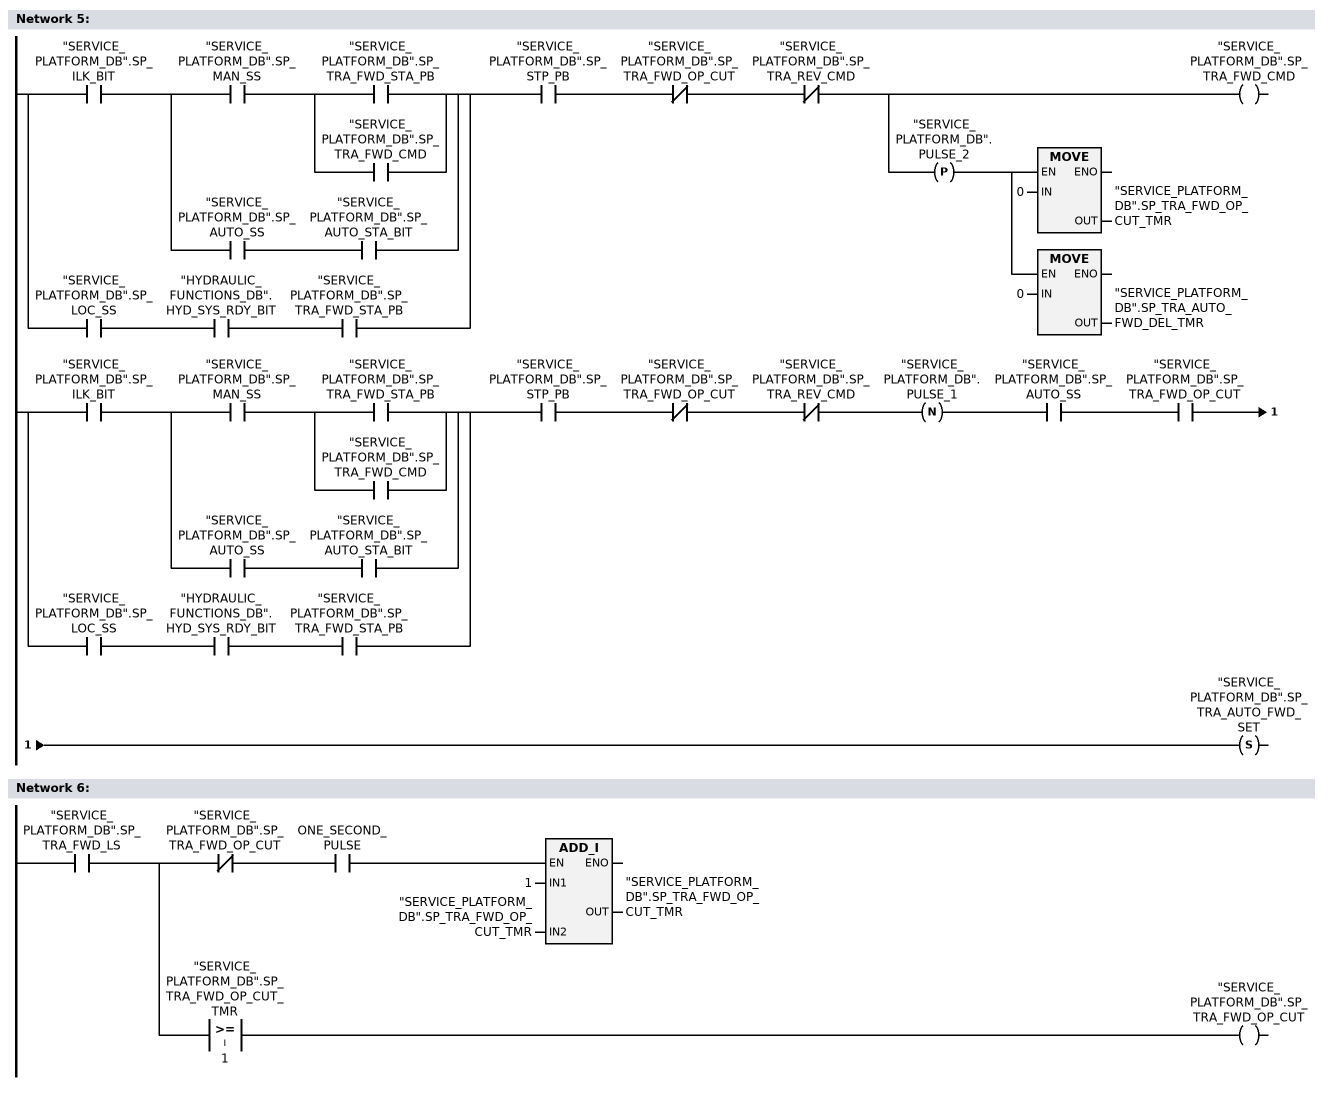
NETWORK
TITLE =
      A(;
      A     "SERVICE_PLATFORM_DB".SP_ILK_BIT;
      A(;
      A     "SERVICE_PLATFORM_DB".SP_MAN_SS;
      A(;
      O     "SERVICE_PLATFORM_DB".SP_TRA_FWD_STA_PB;
      O     "SERVICE_PLATFORM_DB".SP_TRA_FWD_CMD;
      );
      O;
      A     "SERVICE_PLATFORM_DB".SP_AUTO_SS;
      A     "SERVICE_PLATFORM_DB".SP_AUTO_STA_BIT;
      );
      O;
      A     "SERVICE_PLATFORM_DB".SP_LOC_SS;
      A     "HYDRAULIC_FUNCTIONS_DB".HYD_SYS_RDY_BIT;
      A     "SERVICE_PLATFORM_DB".SP_TRA_FWD_STA_PB;
      );
      A     "SERVICE_PLATFORM_DB".SP_STP_PB;
      AN    "SERVICE_PLATFORM_DB".SP_TRA_FWD_OP_CUT;
      AN    "SERVICE_PLATFORM_DB".SP_TRA_REV_CMD;
      =     L 0.0;
      A     L 0.0;
      BLD   102;
      =     "SERVICE_PLATFORM_DB".SP_TRA_FWD_CMD;
      A(;
      A     L 0.0;
      FN    "SERVICE_PLATFORM_DB".PULSE_1;
      );
      A     "SERVICE_PLATFORM_DB".SP_AUTO_SS;
      A     "SERVICE_PLATFORM_DB".SP_TRA_FWD_OP_CUT;
      S     "SERVICE_PLATFORM_DB".SP_TRA_AUTO_FWD_SET;
      A     L 0.0;
      FP    "SERVICE_PLATFORM_DB".PULSE_2;
      =     L 0.1;
      A     L 0.1;
      JNB   M001;
      L     0;
      T     "SERVICE_PLATFORM_DB".SP_TRA_FWD_OP_CUT_TMR;
M001: NOP   0;
      A     L 0.1;
      JNB   M002;
      L     0;
      T     "SERVICE_PLATFORM_DB".SP_TRA_AUTO_FWD_DEL_TMR;
M002: NOP   0;
NETWORK
TITLE =
      A     "SERVICE_PLATFORM_DB".SP_TRA_FWD_LS;
      =     L 0.0;
      A     L 0.0;
      AN    "SERVICE_PLATFORM_DB".SP_TRA_FWD_OP_CUT;
      A     "ONE_SECOND_PULSE";
      JNB   M003;
      L     1;
      L     "SERVICE_PLATFORM_DB".SP_TRA_FWD_OP_CUT_TMR;
      +I;
      T     "SERVICE_PLATFORM_DB".SP_TRA_FWD_OP_CUT_TMR;
M003: NOP   0;
      A     L 0.0;
      A(;
      L     "SERVICE_PLATFORM_DB".SP_TRA_FWD_OP_CUT_TMR;
      L     1;
      >=I;
      );
      =     "SERVICE_PLATFORM_DB".SP_TRA_FWD_OP_CUT;
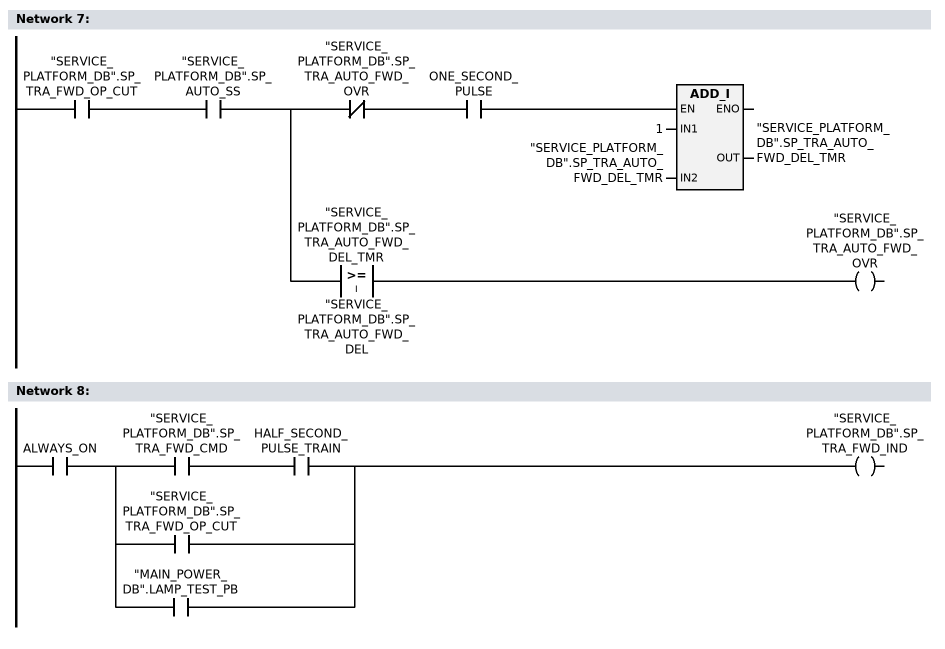
NETWORK
TITLE =
      A     "SERVICE_PLATFORM_DB".SP_TRA_FWD_OP_CUT;
      A     "SERVICE_PLATFORM_DB".SP_AUTO_SS;
      =     L 0.0;
      A     L 0.0;
      AN    "SERVICE_PLATFORM_DB".SP_TRA_AUTO_FWD_OVR;
      A     "ONE_SECOND_PULSE";
      JNB   M004;
      L     1;
      L     "SERVICE_PLATFORM_DB".SP_TRA_AUTO_FWD_DEL_TMR;
      +I;
      T     "SERVICE_PLATFORM_DB".SP_TRA_AUTO_FWD_DEL_TMR;
M004: NOP   0;
      A     L 0.0;
      A(;
      L     "SERVICE_PLATFORM_DB".SP_TRA_AUTO_FWD_DEL_TMR;
      L     "SERVICE_PLATFORM_DB".SP_TRA_AUTO_FWD_DEL;
      >=I;
      );
      =     "SERVICE_PLATFORM_DB".SP_TRA_AUTO_FWD_OVR;
NETWORK
TITLE =
      A     "ALWAYS_ON";
      A(;
      A     "SERVICE_PLATFORM_DB".SP_TRA_FWD_CMD;
      A     "HALF_SECOND_PULSE_TRAIN";
      O     "SERVICE_PLATFORM_DB".SP_TRA_FWD_OP_CUT;
      O     "MAIN_POWER_DB".LAMP_TEST_PB;
      );
      =     "SERVICE_PLATFORM_DB".SP_TRA_FWD_IND;
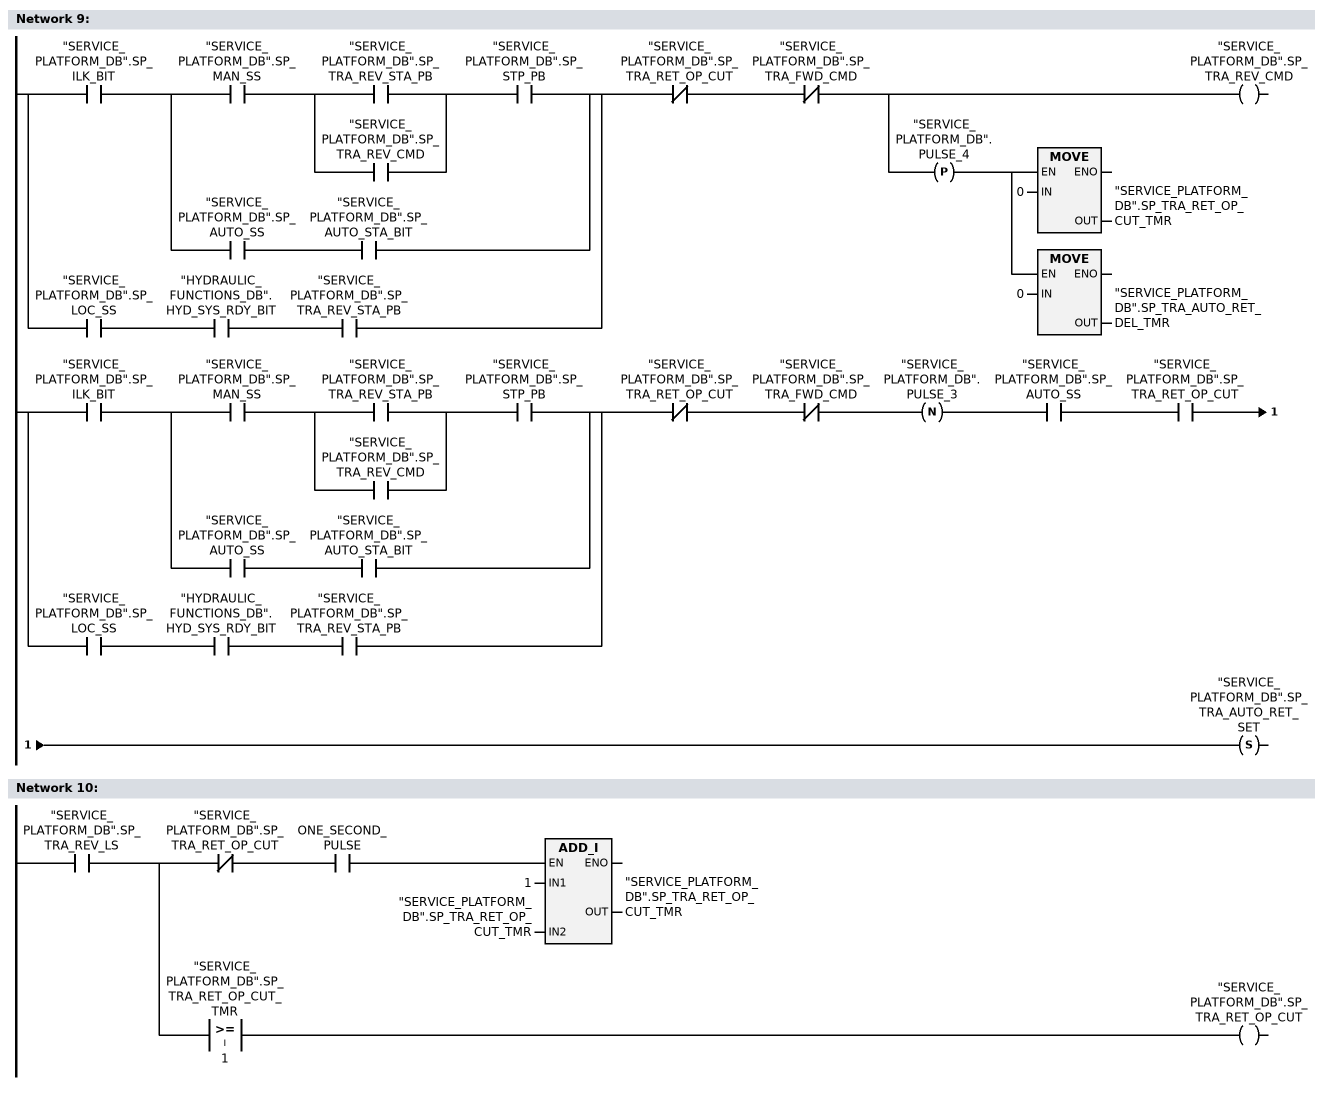
NETWORK
TITLE =
      A(;
      A     "SERVICE_PLATFORM_DB".SP_ILK_BIT;
      A(;
      A     "SERVICE_PLATFORM_DB".SP_MAN_SS;
      A(;
      O     "SERVICE_PLATFORM_DB".SP_TRA_REV_STA_PB;
      O     "SERVICE_PLATFORM_DB".SP_TRA_REV_CMD;
      );
      A     "SERVICE_PLATFORM_DB".SP_STP_PB;
      O;
      A     "SERVICE_PLATFORM_DB".SP_AUTO_SS;
      A     "SERVICE_PLATFORM_DB".SP_AUTO_STA_BIT;
      );
      O;
      A     "SERVICE_PLATFORM_DB".SP_LOC_SS;
      A     "HYDRAULIC_FUNCTIONS_DB".HYD_SYS_RDY_BIT;
      A     "SERVICE_PLATFORM_DB".SP_TRA_REV_STA_PB;
      );
      AN    "SERVICE_PLATFORM_DB".SP_TRA_RET_OP_CUT;
      AN    "SERVICE_PLATFORM_DB".SP_TRA_FWD_CMD;
      =     L 0.0;
      A     L 0.0;
      BLD   102;
      =     "SERVICE_PLATFORM_DB".SP_TRA_REV_CMD;
      A(;
      A     L 0.0;
      FN    "SERVICE_PLATFORM_DB".PULSE_3;
      );
      A     "SERVICE_PLATFORM_DB".SP_AUTO_SS;
      A     "SERVICE_PLATFORM_DB".SP_TRA_RET_OP_CUT;
      S     "SERVICE_PLATFORM_DB".SP_TRA_AUTO_RET_SET;
      A     L 0.0;
      FP    "SERVICE_PLATFORM_DB".PULSE_4;
      =     L 0.1;
      A     L 0.1;
      JNB   M005;
      L     0;
      T     "SERVICE_PLATFORM_DB".SP_TRA_RET_OP_CUT_TMR;
M005: NOP   0;
      A     L 0.1;
      JNB   M006;
      L     0;
      T     "SERVICE_PLATFORM_DB".SP_TRA_AUTO_RET_DEL_TMR;
M006: NOP   0;
NETWORK
TITLE =
      A     "SERVICE_PLATFORM_DB".SP_TRA_REV_LS;
      =     L 0.0;
      A     L 0.0;
      AN    "SERVICE_PLATFORM_DB".SP_TRA_RET_OP_CUT;
      A     "ONE_SECOND_PULSE";
      JNB   M007;
      L     1;
      L     "SERVICE_PLATFORM_DB".SP_TRA_RET_OP_CUT_TMR;
      +I;
      T     "SERVICE_PLATFORM_DB".SP_TRA_RET_OP_CUT_TMR;
M007: NOP   0;
      A     L 0.0;
      A(;
      L     "SERVICE_PLATFORM_DB".SP_TRA_RET_OP_CUT_TMR;
      L     1;
      >=I;
      );
      =     "SERVICE_PLATFORM_DB".SP_TRA_RET_OP_CUT;
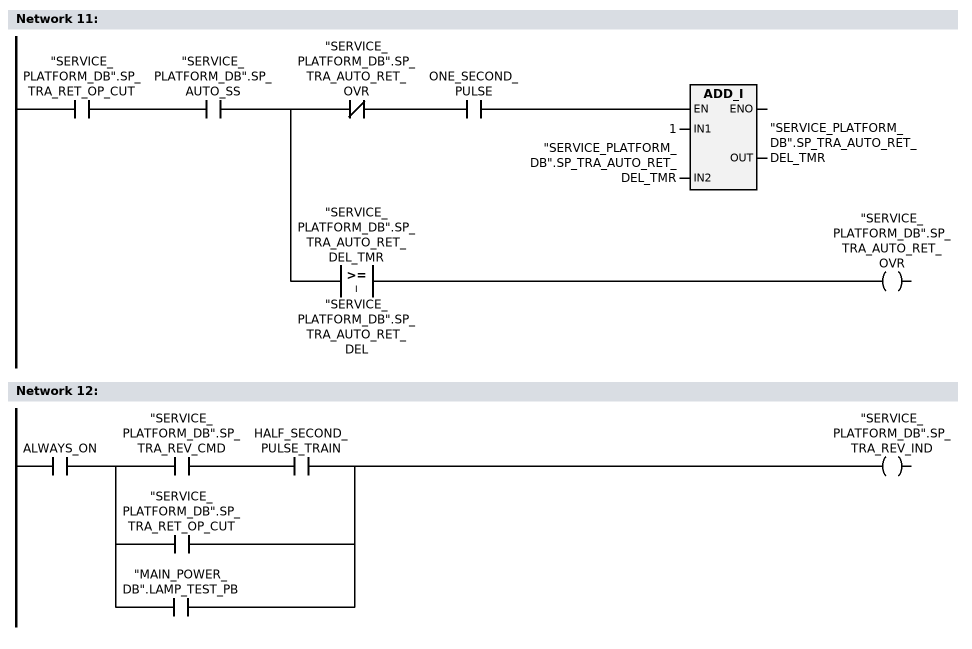
NETWORK
TITLE =
      A     "SERVICE_PLATFORM_DB".SP_TRA_RET_OP_CUT;
      A     "SERVICE_PLATFORM_DB".SP_AUTO_SS;
      =     L 0.0;
      A     L 0.0;
      AN    "SERVICE_PLATFORM_DB".SP_TRA_AUTO_RET_OVR;
      A     "ONE_SECOND_PULSE";
      JNB   M008;
      L     1;
      L     "SERVICE_PLATFORM_DB".SP_TRA_AUTO_RET_DEL_TMR;
      +I;
      T     "SERVICE_PLATFORM_DB".SP_TRA_AUTO_RET_DEL_TMR;
M008: NOP   0;
      A     L 0.0;
      A(;
      L     "SERVICE_PLATFORM_DB".SP_TRA_AUTO_RET_DEL_TMR;
      L     "SERVICE_PLATFORM_DB".SP_TRA_AUTO_RET_DEL;
      >=I;
      );
      =     "SERVICE_PLATFORM_DB".SP_TRA_AUTO_RET_OVR;
NETWORK
TITLE =
      A     "ALWAYS_ON";
      A(;
      A     "SERVICE_PLATFORM_DB".SP_TRA_REV_CMD;
      A     "HALF_SECOND_PULSE_TRAIN";
      O     "SERVICE_PLATFORM_DB".SP_TRA_RET_OP_CUT;
      O     "MAIN_POWER_DB".LAMP_TEST_PB;
      );
      =     "SERVICE_PLATFORM_DB".SP_TRA_REV_IND;
END_FUNCTION

FUNCTION "JAMB_CLEANER" : VOID	// FC 10
AUTHOR : Kamillas
VERSION : 0.1
BEGIN
// (block stored without names or comments; labels and parameter names are numbered)
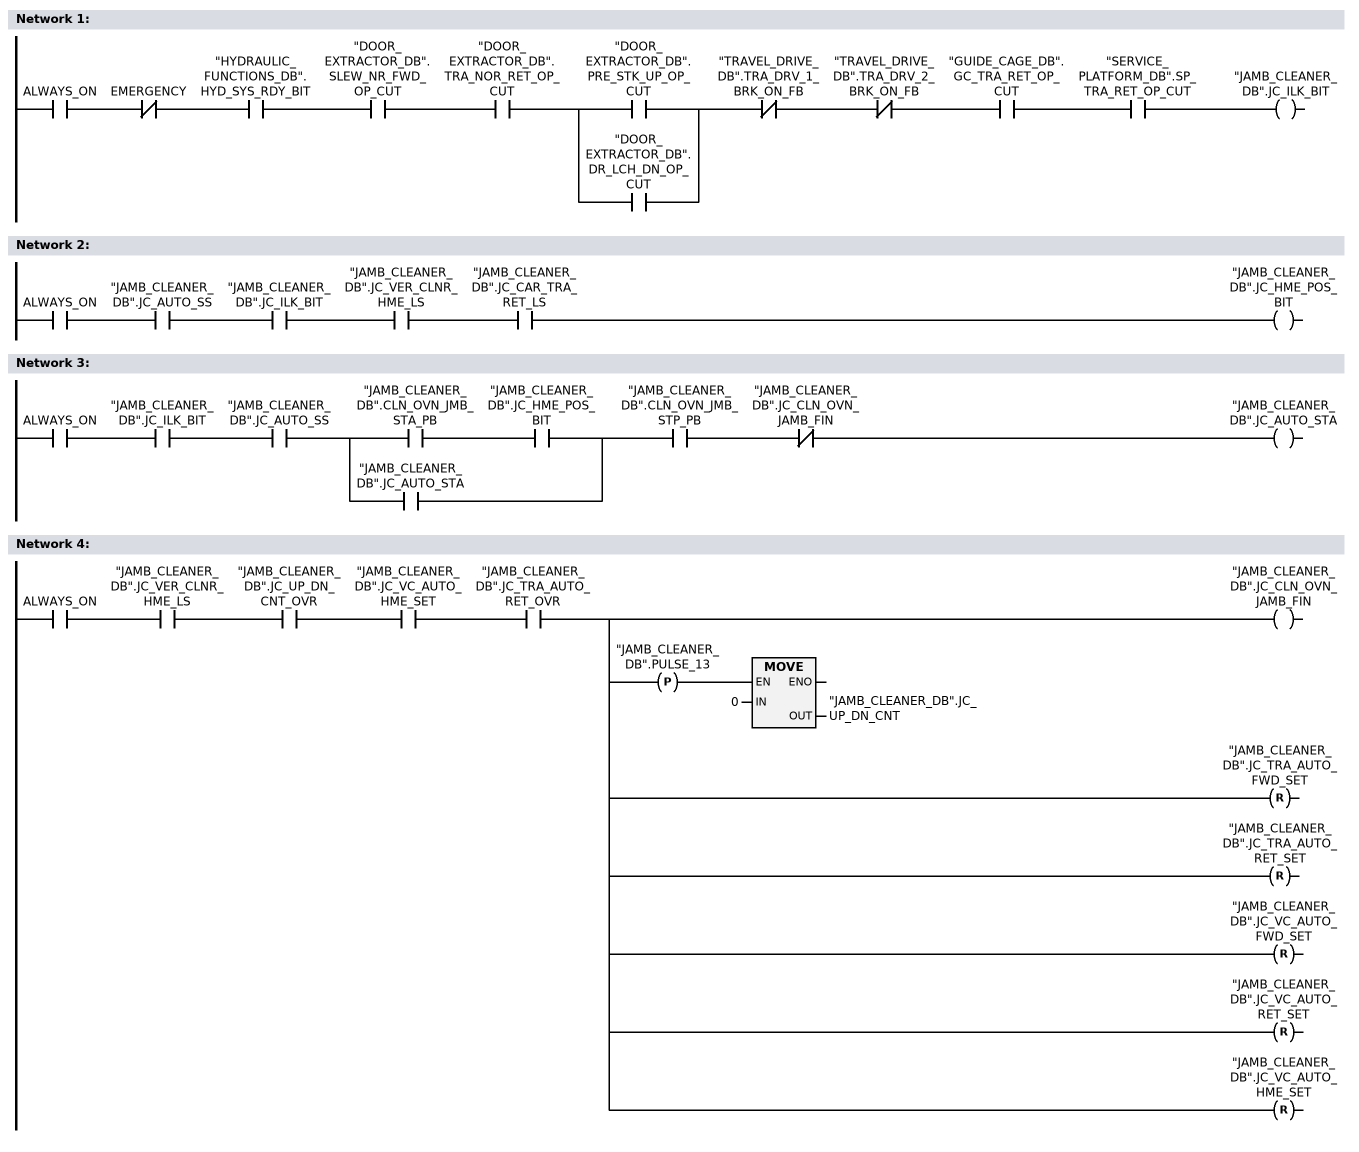
NETWORK
TITLE =
      A     "ALWAYS_ON";
      AN    "EMERGENCY";
      A     "HYDRAULIC_FUNCTIONS_DB".HYD_SYS_RDY_BIT;
      A     "DOOR_EXTRACTOR_DB".SLEW_NR_FWD_OP_CUT;
      A     "DOOR_EXTRACTOR_DB".TRA_NOR_RET_OP_CUT;
      A(;
      O     "DOOR_EXTRACTOR_DB".PRE_STK_UP_OP_CUT;
      O     "DOOR_EXTRACTOR_DB".DR_LCH_DN_OP_CUT;
      );
      AN    "TRAVEL_DRIVE_DB".TRA_DRV_1_BRK_ON_FB;
      AN    "TRAVEL_DRIVE_DB".TRA_DRV_2_BRK_ON_FB;
      A     "GUIDE_CAGE_DB".GC_TRA_RET_OP_CUT;
      A     "SERVICE_PLATFORM_DB".SP_TRA_RET_OP_CUT;
      =     "JAMB_CLEANER_DB".JC_ILK_BIT;
NETWORK
TITLE =
      A     "ALWAYS_ON";
      A     "JAMB_CLEANER_DB".JC_AUTO_SS;
      A     "JAMB_CLEANER_DB".JC_ILK_BIT;
      A     "JAMB_CLEANER_DB".JC_VER_CLNR_HME_LS;
      A     "JAMB_CLEANER_DB".JC_CAR_TRA_RET_LS;
      =     "JAMB_CLEANER_DB".JC_HME_POS_BIT;
NETWORK
TITLE =
      A     "ALWAYS_ON";
      A     "JAMB_CLEANER_DB".JC_ILK_BIT;
      A     "JAMB_CLEANER_DB".JC_AUTO_SS;
      A(;
      A     "JAMB_CLEANER_DB".CLN_OVN_JMB_STA_PB;
      A     "JAMB_CLEANER_DB".JC_HME_POS_BIT;
      O     "JAMB_CLEANER_DB".JC_AUTO_STA;
      );
      A     "JAMB_CLEANER_DB".CLN_OVN_JMB_STP_PB;
      AN    "JAMB_CLEANER_DB".JC_CLN_OVN_JAMB_FIN;
      =     "JAMB_CLEANER_DB".JC_AUTO_STA;
NETWORK
TITLE =
      A     "ALWAYS_ON";
      A     "JAMB_CLEANER_DB".JC_VER_CLNR_HME_LS;
      A     "JAMB_CLEANER_DB".JC_UP_DN_CNT_OVR;
      A     "JAMB_CLEANER_DB".JC_VC_AUTO_HME_SET;
      A     "JAMB_CLEANER_DB".JC_TRA_AUTO_RET_OVR;
      =     L 0.0;
      A     L 0.0;
      BLD   102;
      =     "JAMB_CLEANER_DB".JC_CLN_OVN_JAMB_FIN;
      A     L 0.0;
      FP    "JAMB_CLEANER_DB".PULSE_13;
      JNB   M001;
      L     0;
      T     "JAMB_CLEANER_DB".JC_UP_DN_CNT;
M001: NOP   0;
      A     L 0.0;
      BLD   102;
      R     "JAMB_CLEANER_DB".JC_TRA_AUTO_FWD_SET;
      A     L 0.0;
      BLD   102;
      R     "JAMB_CLEANER_DB".JC_TRA_AUTO_RET_SET;
      A     L 0.0;
      BLD   102;
      R     "JAMB_CLEANER_DB".JC_VC_AUTO_FWD_SET;
      A     L 0.0;
      BLD   102;
      R     "JAMB_CLEANER_DB".JC_VC_AUTO_RET_SET;
      A     L 0.0;
      BLD   102;
      R     "JAMB_CLEANER_DB".JC_VC_AUTO_HME_SET;
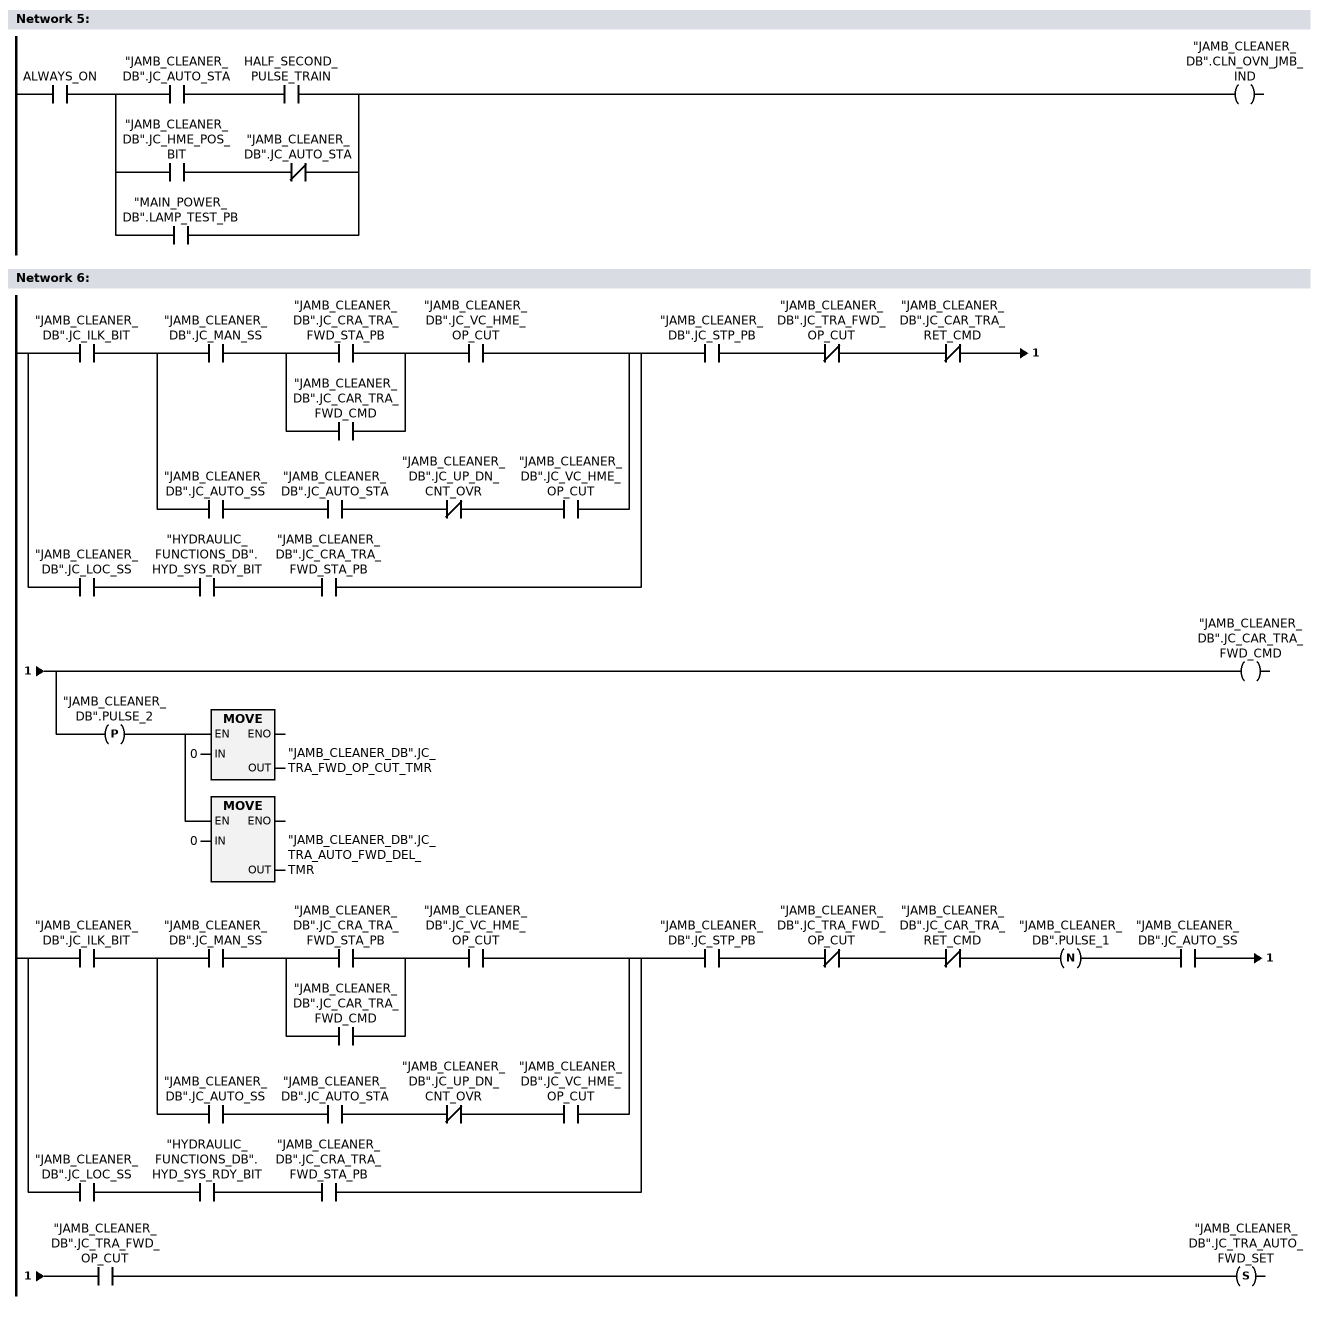
NETWORK
TITLE =
      A     "ALWAYS_ON";
      A(;
      A     "JAMB_CLEANER_DB".JC_AUTO_STA;
      A     "HALF_SECOND_PULSE_TRAIN";
      O;
      A     "JAMB_CLEANER_DB".JC_HME_POS_BIT;
      AN    "JAMB_CLEANER_DB".JC_AUTO_STA;
      O     "MAIN_POWER_DB".LAMP_TEST_PB;
      );
      =     "JAMB_CLEANER_DB".CLN_OVN_JMB_IND;
NETWORK
TITLE =
      A(;
      A     "JAMB_CLEANER_DB".JC_ILK_BIT;
      A(;
      A     "JAMB_CLEANER_DB".JC_MAN_SS;
      A(;
      O     "JAMB_CLEANER_DB".JC_CRA_TRA_FWD_STA_PB;
      O     "JAMB_CLEANER_DB".JC_CAR_TRA_FWD_CMD;
      );
      A     "JAMB_CLEANER_DB".JC_VC_HME_OP_CUT;
      O;
      A     "JAMB_CLEANER_DB".JC_AUTO_SS;
      A     "JAMB_CLEANER_DB".JC_AUTO_STA;
      AN    "JAMB_CLEANER_DB".JC_UP_DN_CNT_OVR;
      A     "JAMB_CLEANER_DB".JC_VC_HME_OP_CUT;
      );
      O;
      A     "JAMB_CLEANER_DB".JC_LOC_SS;
      A     "HYDRAULIC_FUNCTIONS_DB".HYD_SYS_RDY_BIT;
      A     "JAMB_CLEANER_DB".JC_CRA_TRA_FWD_STA_PB;
      );
      A     "JAMB_CLEANER_DB".JC_STP_PB;
      AN    "JAMB_CLEANER_DB".JC_TRA_FWD_OP_CUT;
      AN    "JAMB_CLEANER_DB".JC_CAR_TRA_RET_CMD;
      =     L 0.0;
      A     L 0.0;
      BLD   102;
      =     "JAMB_CLEANER_DB".JC_CAR_TRA_FWD_CMD;
      A(;
      A     L 0.0;
      FN    "JAMB_CLEANER_DB".PULSE_1;
      );
      A     "JAMB_CLEANER_DB".JC_AUTO_SS;
      A     "JAMB_CLEANER_DB".JC_TRA_FWD_OP_CUT;
      S     "JAMB_CLEANER_DB".JC_TRA_AUTO_FWD_SET;
      A     L 0.0;
      FP    "JAMB_CLEANER_DB".PULSE_2;
      =     L 0.1;
      A     L 0.1;
      JNB   M002;
      L     0;
      T     "JAMB_CLEANER_DB".JC_TRA_FWD_OP_CUT_TMR;
M002: NOP   0;
      A     L 0.1;
      JNB   M003;
      L     0;
      T     "JAMB_CLEANER_DB".JC_TRA_AUTO_FWD_DEL_TMR;
M003: NOP   0;
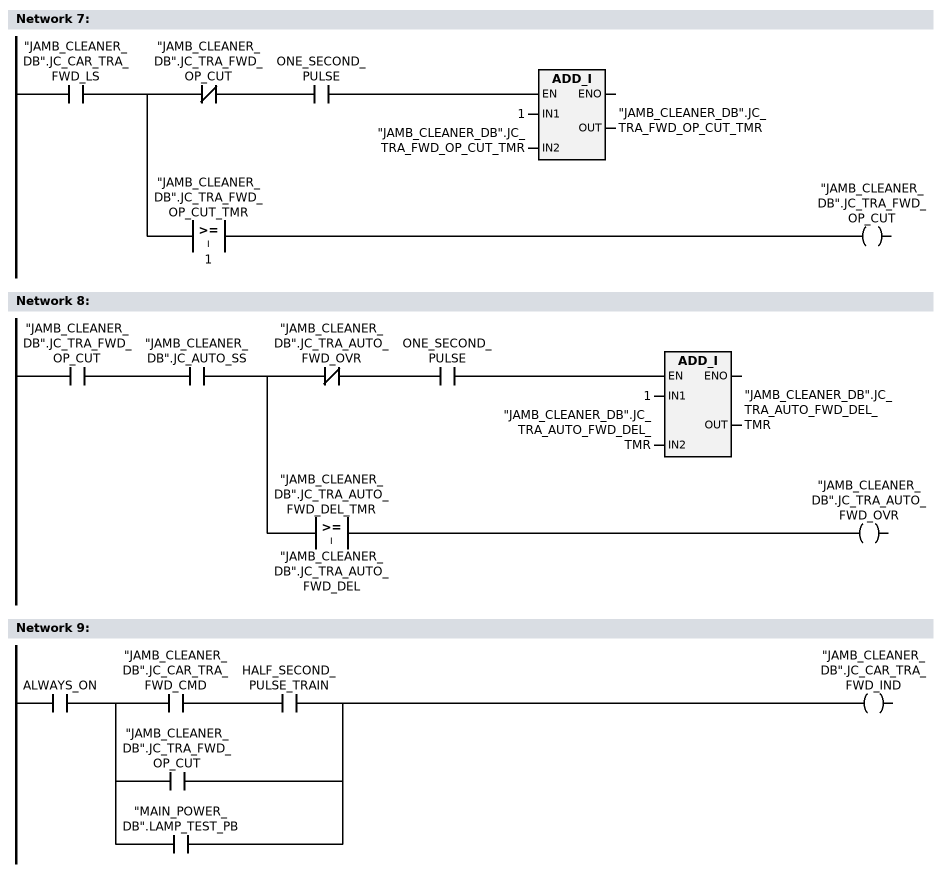
NETWORK
TITLE =
      A     "JAMB_CLEANER_DB".JC_CAR_TRA_FWD_LS;
      =     L 0.0;
      A     L 0.0;
      AN    "JAMB_CLEANER_DB".JC_TRA_FWD_OP_CUT;
      A     "ONE_SECOND_PULSE";
      JNB   M004;
      L     1;
      L     "JAMB_CLEANER_DB".JC_TRA_FWD_OP_CUT_TMR;
      +I;
      T     "JAMB_CLEANER_DB".JC_TRA_FWD_OP_CUT_TMR;
M004: NOP   0;
      A     L 0.0;
      A(;
      L     "JAMB_CLEANER_DB".JC_TRA_FWD_OP_CUT_TMR;
      L     1;
      >=I;
      );
      =     "JAMB_CLEANER_DB".JC_TRA_FWD_OP_CUT;
NETWORK
TITLE =
      A     "JAMB_CLEANER_DB".JC_TRA_FWD_OP_CUT;
      A     "JAMB_CLEANER_DB".JC_AUTO_SS;
      =     L 0.0;
      A     L 0.0;
      AN    "JAMB_CLEANER_DB".JC_TRA_AUTO_FWD_OVR;
      A     "ONE_SECOND_PULSE";
      JNB   M005;
      L     1;
      L     "JAMB_CLEANER_DB".JC_TRA_AUTO_FWD_DEL_TMR;
      +I;
      T     "JAMB_CLEANER_DB".JC_TRA_AUTO_FWD_DEL_TMR;
M005: NOP   0;
      A     L 0.0;
      A(;
      L     "JAMB_CLEANER_DB".JC_TRA_AUTO_FWD_DEL_TMR;
      L     "JAMB_CLEANER_DB".JC_TRA_AUTO_FWD_DEL;
      >=I;
      );
      =     "JAMB_CLEANER_DB".JC_TRA_AUTO_FWD_OVR;
NETWORK
TITLE =
      A     "ALWAYS_ON";
      A(;
      A     "JAMB_CLEANER_DB".JC_CAR_TRA_FWD_CMD;
      A     "HALF_SECOND_PULSE_TRAIN";
      O     "JAMB_CLEANER_DB".JC_TRA_FWD_OP_CUT;
      O     "MAIN_POWER_DB".LAMP_TEST_PB;
      );
      =     "JAMB_CLEANER_DB".JC_CAR_TRA_FWD_IND;
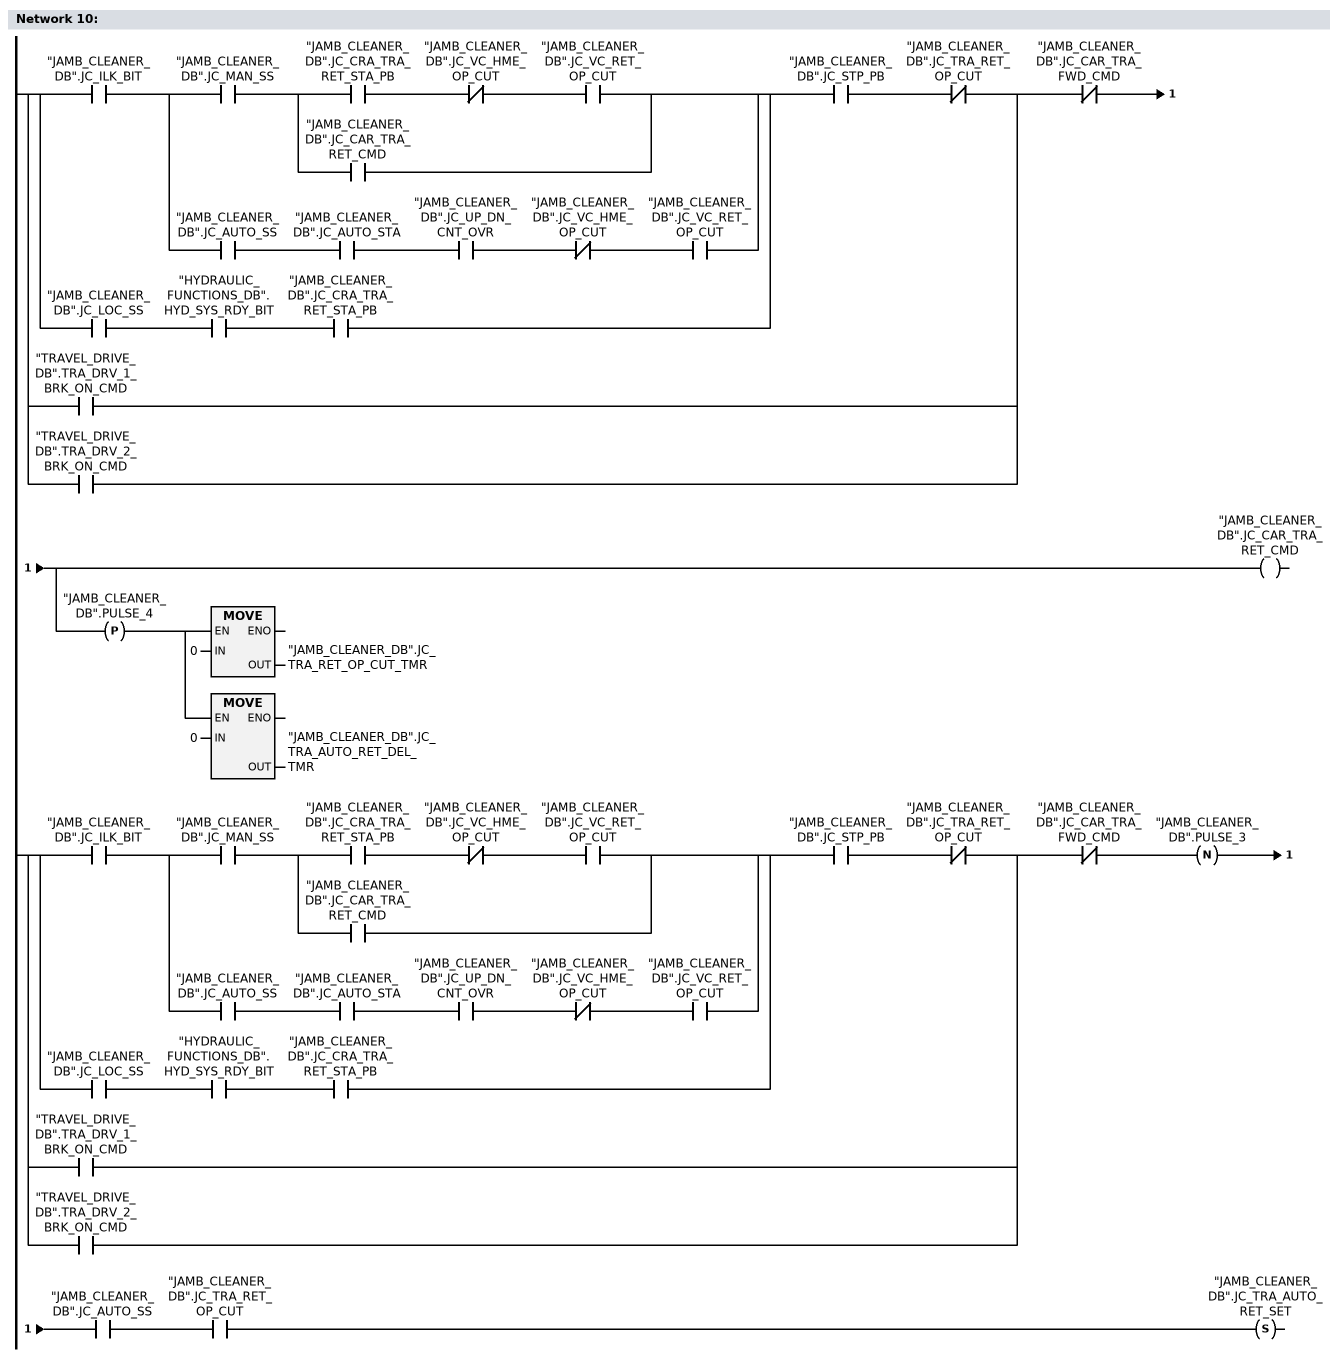
NETWORK
TITLE =
      A(;
      A(;
      A     "JAMB_CLEANER_DB".JC_ILK_BIT;
      A(;
      A     "JAMB_CLEANER_DB".JC_MAN_SS;
      A(;
      A     "JAMB_CLEANER_DB".JC_CRA_TRA_RET_STA_PB;
      AN    "JAMB_CLEANER_DB".JC_VC_HME_OP_CUT;
      A     "JAMB_CLEANER_DB".JC_VC_RET_OP_CUT;
      O     "JAMB_CLEANER_DB".JC_CAR_TRA_RET_CMD;
      );
      O;
      A     "JAMB_CLEANER_DB".JC_AUTO_SS;
      A     "JAMB_CLEANER_DB".JC_AUTO_STA;
      A     "JAMB_CLEANER_DB".JC_UP_DN_CNT_OVR;
      AN    "JAMB_CLEANER_DB".JC_VC_HME_OP_CUT;
      A     "JAMB_CLEANER_DB".JC_VC_RET_OP_CUT;
      );
      O;
      A     "JAMB_CLEANER_DB".JC_LOC_SS;
      A     "HYDRAULIC_FUNCTIONS_DB".HYD_SYS_RDY_BIT;
      A     "JAMB_CLEANER_DB".JC_CRA_TRA_RET_STA_PB;
      );
      A     "JAMB_CLEANER_DB".JC_STP_PB;
      AN    "JAMB_CLEANER_DB".JC_TRA_RET_OP_CUT;
      O     "TRAVEL_DRIVE_DB".TRA_DRV_1_BRK_ON_CMD;
      O     "TRAVEL_DRIVE_DB".TRA_DRV_2_BRK_ON_CMD;
      );
      AN    "JAMB_CLEANER_DB".JC_CAR_TRA_FWD_CMD;
      =     L 0.0;
      A     L 0.0;
      BLD   102;
      =     "JAMB_CLEANER_DB".JC_CAR_TRA_RET_CMD;
      A(;
      A     L 0.0;
      FN    "JAMB_CLEANER_DB".PULSE_3;
      );
      A     "JAMB_CLEANER_DB".JC_AUTO_SS;
      A     "JAMB_CLEANER_DB".JC_TRA_RET_OP_CUT;
      S     "JAMB_CLEANER_DB".JC_TRA_AUTO_RET_SET;
      A     L 0.0;
      FP    "JAMB_CLEANER_DB".PULSE_4;
      =     L 0.1;
      A     L 0.1;
      JNB   M006;
      L     0;
      T     "JAMB_CLEANER_DB".JC_TRA_RET_OP_CUT_TMR;
M006: NOP   0;
      A     L 0.1;
      JNB   M007;
      L     0;
      T     "JAMB_CLEANER_DB".JC_TRA_AUTO_RET_DEL_TMR;
M007: NOP   0;
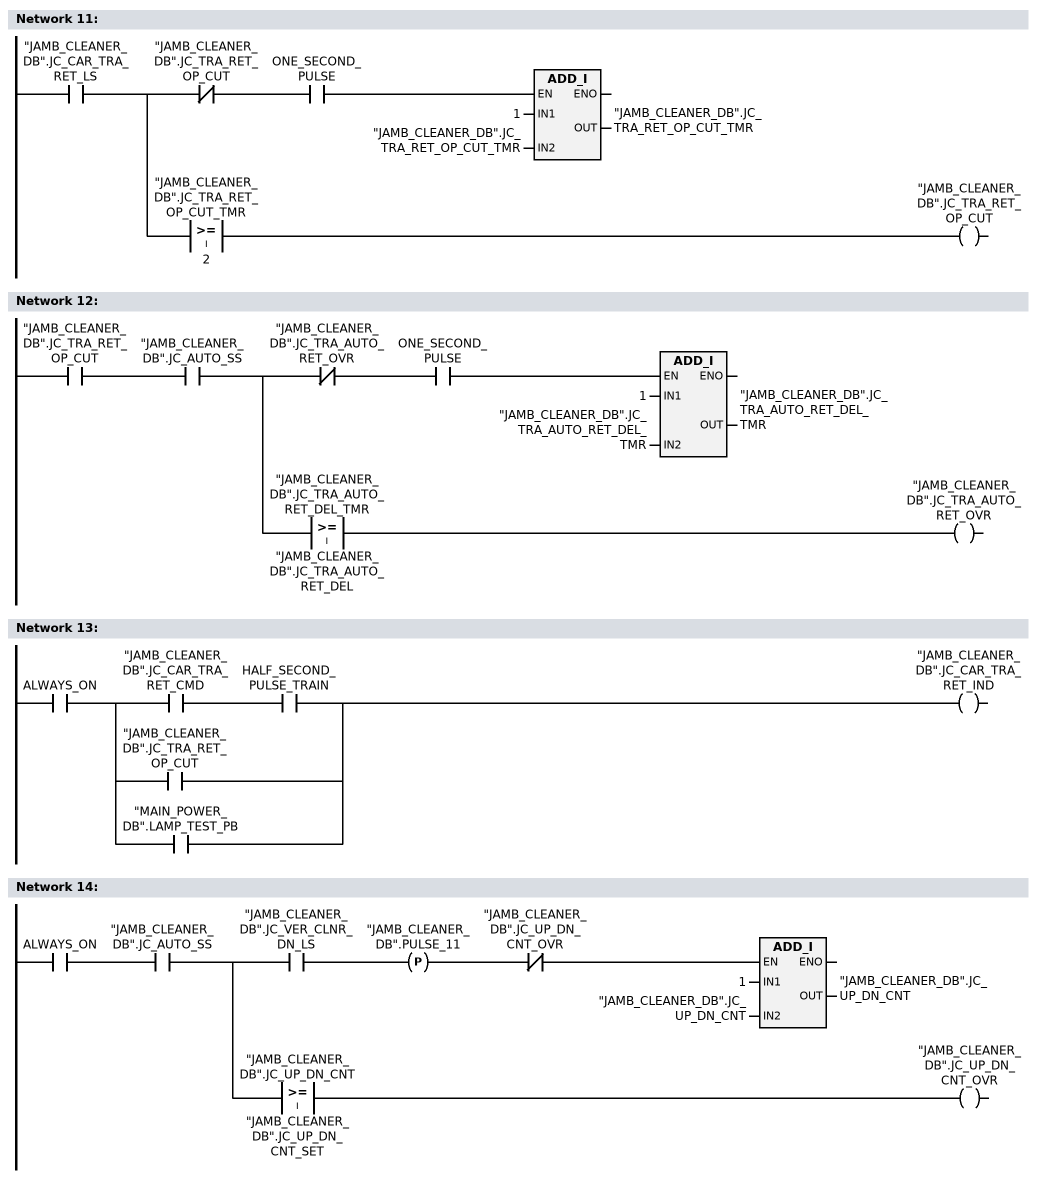
NETWORK
TITLE =
      A     "JAMB_CLEANER_DB".JC_CAR_TRA_RET_LS;
      =     L 0.0;
      A     L 0.0;
      AN    "JAMB_CLEANER_DB".JC_TRA_RET_OP_CUT;
      A     "ONE_SECOND_PULSE";
      JNB   M008;
      L     1;
      L     "JAMB_CLEANER_DB".JC_TRA_RET_OP_CUT_TMR;
      +I;
      T     "JAMB_CLEANER_DB".JC_TRA_RET_OP_CUT_TMR;
M008: NOP   0;
      A     L 0.0;
      A(;
      L     "JAMB_CLEANER_DB".JC_TRA_RET_OP_CUT_TMR;
      L     2;
      >=I;
      );
      =     "JAMB_CLEANER_DB".JC_TRA_RET_OP_CUT;
NETWORK
TITLE =
      A     "JAMB_CLEANER_DB".JC_TRA_RET_OP_CUT;
      A     "JAMB_CLEANER_DB".JC_AUTO_SS;
      =     L 0.0;
      A     L 0.0;
      AN    "JAMB_CLEANER_DB".JC_TRA_AUTO_RET_OVR;
      A     "ONE_SECOND_PULSE";
      JNB   M009;
      L     1;
      L     "JAMB_CLEANER_DB".JC_TRA_AUTO_RET_DEL_TMR;
      +I;
      T     "JAMB_CLEANER_DB".JC_TRA_AUTO_RET_DEL_TMR;
M009: NOP   0;
      A     L 0.0;
      A(;
      L     "JAMB_CLEANER_DB".JC_TRA_AUTO_RET_DEL_TMR;
      L     "JAMB_CLEANER_DB".JC_TRA_AUTO_RET_DEL;
      >=I;
      );
      =     "JAMB_CLEANER_DB".JC_TRA_AUTO_RET_OVR;
NETWORK
TITLE =
      A     "ALWAYS_ON";
      A(;
      A     "JAMB_CLEANER_DB".JC_CAR_TRA_RET_CMD;
      A     "HALF_SECOND_PULSE_TRAIN";
      O     "JAMB_CLEANER_DB".JC_TRA_RET_OP_CUT;
      O     "MAIN_POWER_DB".LAMP_TEST_PB;
      );
      =     "JAMB_CLEANER_DB".JC_CAR_TRA_RET_IND;
NETWORK
TITLE =
      A     "ALWAYS_ON";
      A     "JAMB_CLEANER_DB".JC_AUTO_SS;
      =     L 0.0;
      A     L 0.0;
      A     "JAMB_CLEANER_DB".JC_VER_CLNR_DN_LS;
      FP    "JAMB_CLEANER_DB".PULSE_11;
      AN    "JAMB_CLEANER_DB".JC_UP_DN_CNT_OVR;
      JNB   M010;
      L     1;
      L     "JAMB_CLEANER_DB".JC_UP_DN_CNT;
      +I;
      T     "JAMB_CLEANER_DB".JC_UP_DN_CNT;
M010: NOP   0;
      A     L 0.0;
      A(;
      L     "JAMB_CLEANER_DB".JC_UP_DN_CNT;
      L     "JAMB_CLEANER_DB".JC_UP_DN_CNT_SET;
      >=I;
      );
      =     "JAMB_CLEANER_DB".JC_UP_DN_CNT_OVR;
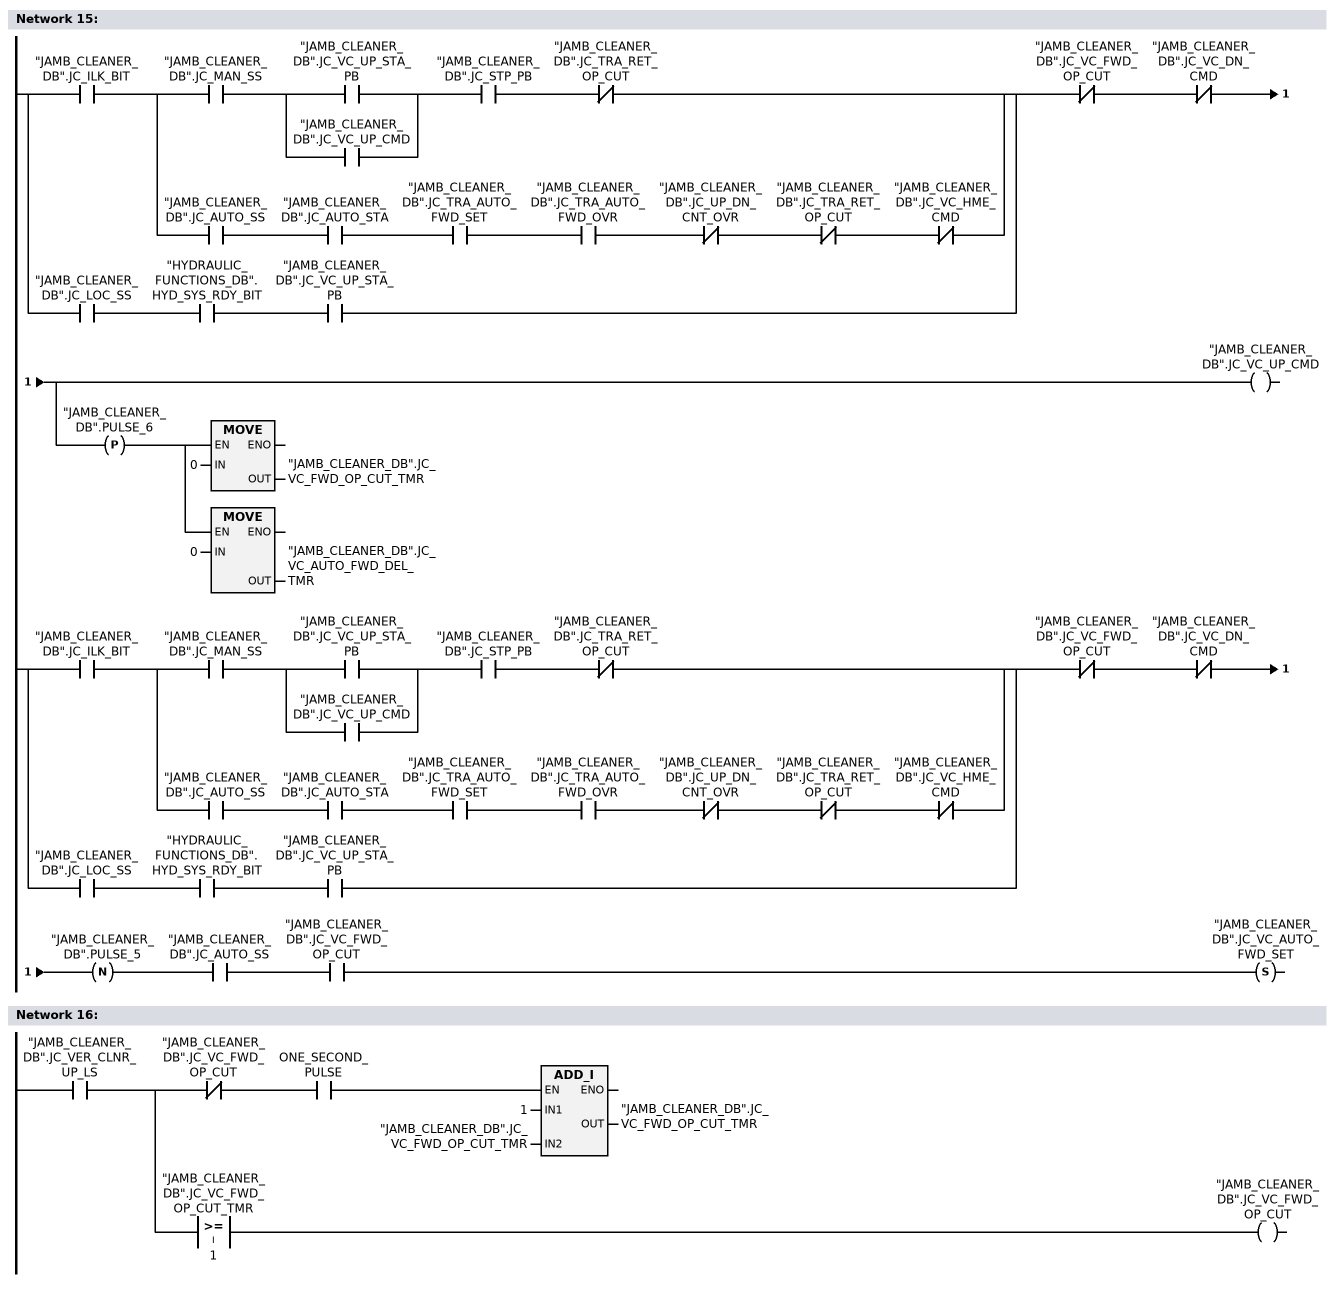
NETWORK
TITLE =
      A(;
      A     "JAMB_CLEANER_DB".JC_ILK_BIT;
      A(;
      A     "JAMB_CLEANER_DB".JC_MAN_SS;
      A(;
      O     "JAMB_CLEANER_DB".JC_VC_UP_STA_PB;
      O     "JAMB_CLEANER_DB".JC_VC_UP_CMD;
      );
      A     "JAMB_CLEANER_DB".JC_STP_PB;
      AN    "JAMB_CLEANER_DB".JC_TRA_RET_OP_CUT;
      O;
      A     "JAMB_CLEANER_DB".JC_AUTO_SS;
      A     "JAMB_CLEANER_DB".JC_AUTO_STA;
      A     "JAMB_CLEANER_DB".JC_TRA_AUTO_FWD_SET;
      A     "JAMB_CLEANER_DB".JC_TRA_AUTO_FWD_OVR;
      AN    "JAMB_CLEANER_DB".JC_UP_DN_CNT_OVR;
      AN    "JAMB_CLEANER_DB".JC_TRA_RET_OP_CUT;
      AN    "JAMB_CLEANER_DB".JC_VC_HME_CMD;
      );
      O;
      A     "JAMB_CLEANER_DB".JC_LOC_SS;
      A     "HYDRAULIC_FUNCTIONS_DB".HYD_SYS_RDY_BIT;
      A     "JAMB_CLEANER_DB".JC_VC_UP_STA_PB;
      );
      AN    "JAMB_CLEANER_DB".JC_VC_FWD_OP_CUT;
      AN    "JAMB_CLEANER_DB".JC_VC_DN_CMD;
      =     L 0.0;
      A     L 0.0;
      BLD   102;
      =     "JAMB_CLEANER_DB".JC_VC_UP_CMD;
      A(;
      A     L 0.0;
      FN    "JAMB_CLEANER_DB".PULSE_5;
      );
      A     "JAMB_CLEANER_DB".JC_AUTO_SS;
      A     "JAMB_CLEANER_DB".JC_VC_FWD_OP_CUT;
      S     "JAMB_CLEANER_DB".JC_VC_AUTO_FWD_SET;
      A     L 0.0;
      FP    "JAMB_CLEANER_DB".PULSE_6;
      =     L 0.1;
      A     L 0.1;
      JNB   M011;
      L     0;
      T     "JAMB_CLEANER_DB".JC_VC_FWD_OP_CUT_TMR;
M011: NOP   0;
      A     L 0.1;
      JNB   M012;
      L     0;
      T     "JAMB_CLEANER_DB".JC_VC_AUTO_FWD_DEL_TMR;
M012: NOP   0;
NETWORK
TITLE =
      A     "JAMB_CLEANER_DB".JC_VER_CLNR_UP_LS;
      =     L 0.0;
      A     L 0.0;
      AN    "JAMB_CLEANER_DB".JC_VC_FWD_OP_CUT;
      A     "ONE_SECOND_PULSE";
      JNB   M013;
      L     1;
      L     "JAMB_CLEANER_DB".JC_VC_FWD_OP_CUT_TMR;
      +I;
      T     "JAMB_CLEANER_DB".JC_VC_FWD_OP_CUT_TMR;
M013: NOP   0;
      A     L 0.0;
      A(;
      L     "JAMB_CLEANER_DB".JC_VC_FWD_OP_CUT_TMR;
      L     1;
      >=I;
      );
      =     "JAMB_CLEANER_DB".JC_VC_FWD_OP_CUT;
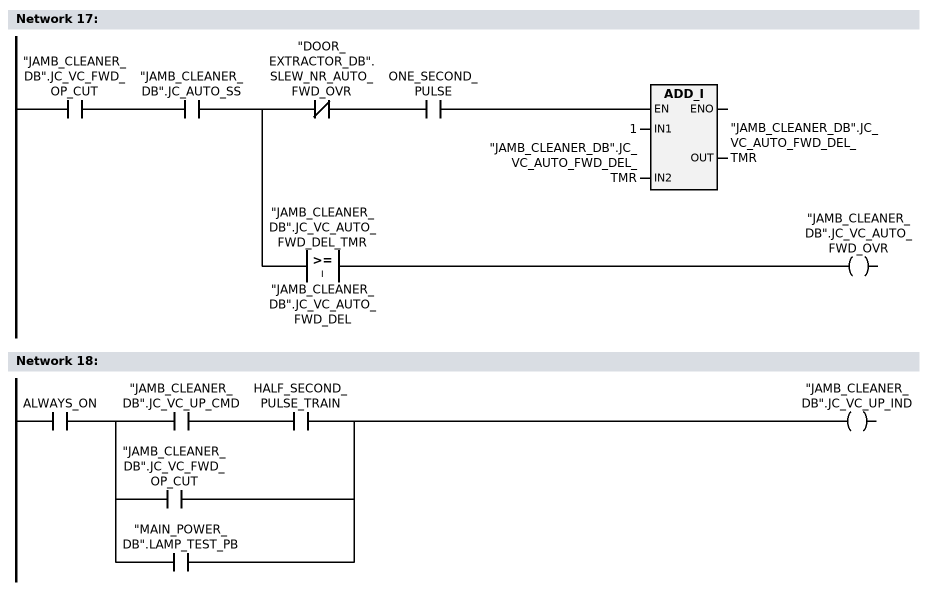
NETWORK
TITLE =
      A     "JAMB_CLEANER_DB".JC_VC_FWD_OP_CUT;
      A     "JAMB_CLEANER_DB".JC_AUTO_SS;
      =     L 0.0;
      A     L 0.0;
      AN    "DOOR_EXTRACTOR_DB".SLEW_NR_AUTO_FWD_OVR;
      A     "ONE_SECOND_PULSE";
      JNB   M014;
      L     1;
      L     "JAMB_CLEANER_DB".JC_VC_AUTO_FWD_DEL_TMR;
      +I;
      T     "JAMB_CLEANER_DB".JC_VC_AUTO_FWD_DEL_TMR;
M014: NOP   0;
      A     L 0.0;
      A(;
      L     "JAMB_CLEANER_DB".JC_VC_AUTO_FWD_DEL_TMR;
      L     "JAMB_CLEANER_DB".JC_VC_AUTO_FWD_DEL;
      >=I;
      );
      =     "JAMB_CLEANER_DB".JC_VC_AUTO_FWD_OVR;
NETWORK
TITLE =
      A     "ALWAYS_ON";
      A(;
      A     "JAMB_CLEANER_DB".JC_VC_UP_CMD;
      A     "HALF_SECOND_PULSE_TRAIN";
      O     "JAMB_CLEANER_DB".JC_VC_FWD_OP_CUT;
      O     "MAIN_POWER_DB".LAMP_TEST_PB;
      );
      =     "JAMB_CLEANER_DB".JC_VC_UP_IND;
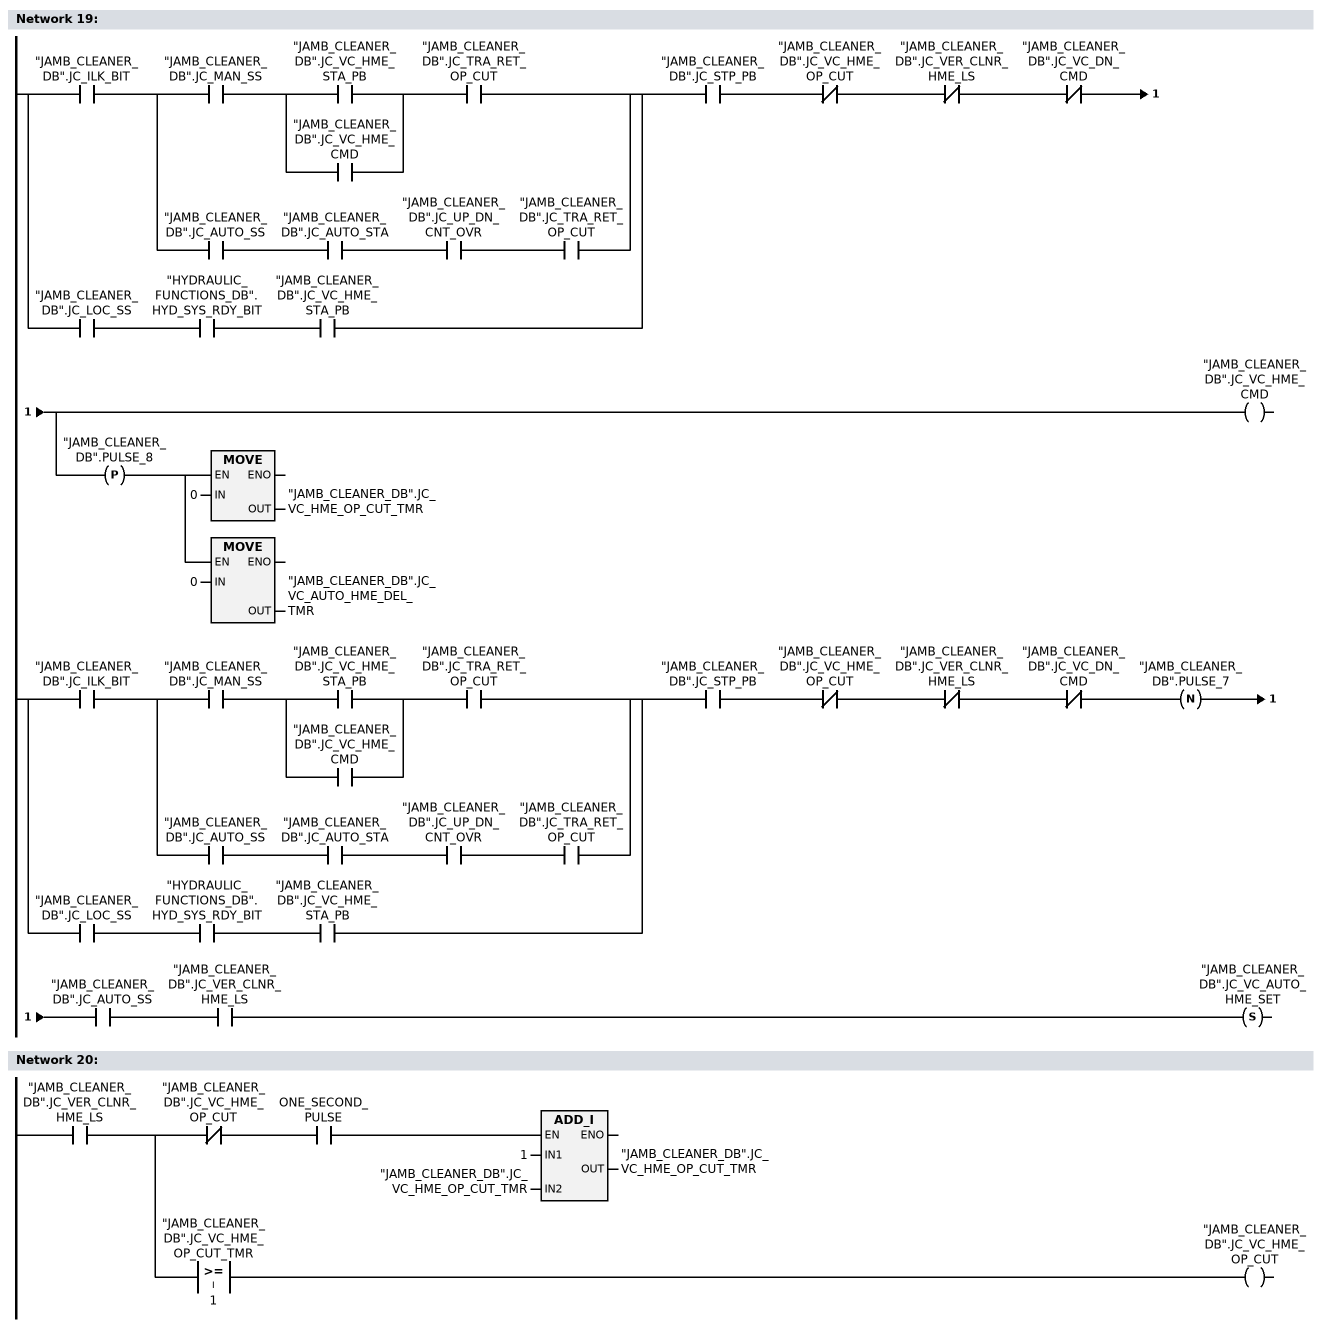
NETWORK
TITLE =
      A(;
      A     "JAMB_CLEANER_DB".JC_ILK_BIT;
      A(;
      A     "JAMB_CLEANER_DB".JC_MAN_SS;
      A(;
      O     "JAMB_CLEANER_DB".JC_VC_HME_STA_PB;
      O     "JAMB_CLEANER_DB".JC_VC_HME_CMD;
      );
      A     "JAMB_CLEANER_DB".JC_TRA_RET_OP_CUT;
      O;
      A     "JAMB_CLEANER_DB".JC_AUTO_SS;
      A     "JAMB_CLEANER_DB".JC_AUTO_STA;
      A     "JAMB_CLEANER_DB".JC_UP_DN_CNT_OVR;
      A     "JAMB_CLEANER_DB".JC_TRA_RET_OP_CUT;
      );
      O;
      A     "JAMB_CLEANER_DB".JC_LOC_SS;
      A     "HYDRAULIC_FUNCTIONS_DB".HYD_SYS_RDY_BIT;
      A     "JAMB_CLEANER_DB".JC_VC_HME_STA_PB;
      );
      A     "JAMB_CLEANER_DB".JC_STP_PB;
      AN    "JAMB_CLEANER_DB".JC_VC_HME_OP_CUT;
      AN    "JAMB_CLEANER_DB".JC_VER_CLNR_HME_LS;
      AN    "JAMB_CLEANER_DB".JC_VC_DN_CMD;
      =     L 0.0;
      A     L 0.0;
      BLD   102;
      =     "JAMB_CLEANER_DB".JC_VC_HME_CMD;
      A(;
      A     L 0.0;
      FN    "JAMB_CLEANER_DB".PULSE_7;
      );
      A     "JAMB_CLEANER_DB".JC_AUTO_SS;
      A     "JAMB_CLEANER_DB".JC_VER_CLNR_HME_LS;
      S     "JAMB_CLEANER_DB".JC_VC_AUTO_HME_SET;
      A     L 0.0;
      FP    "JAMB_CLEANER_DB".PULSE_8;
      =     L 0.1;
      A     L 0.1;
      JNB   M015;
      L     0;
      T     "JAMB_CLEANER_DB".JC_VC_HME_OP_CUT_TMR;
M015: NOP   0;
      A     L 0.1;
      JNB   M016;
      L     0;
      T     "JAMB_CLEANER_DB".JC_VC_AUTO_HME_DEL_TMR;
M016: NOP   0;
NETWORK
TITLE =
      A     "JAMB_CLEANER_DB".JC_VER_CLNR_HME_LS;
      =     L 0.0;
      A     L 0.0;
      AN    "JAMB_CLEANER_DB".JC_VC_HME_OP_CUT;
      A     "ONE_SECOND_PULSE";
      JNB   M017;
      L     1;
      L     "JAMB_CLEANER_DB".JC_VC_HME_OP_CUT_TMR;
      +I;
      T     "JAMB_CLEANER_DB".JC_VC_HME_OP_CUT_TMR;
M017: NOP   0;
      A     L 0.0;
      A(;
      L     "JAMB_CLEANER_DB".JC_VC_HME_OP_CUT_TMR;
      L     1;
      >=I;
      );
      =     "JAMB_CLEANER_DB".JC_VC_HME_OP_CUT;
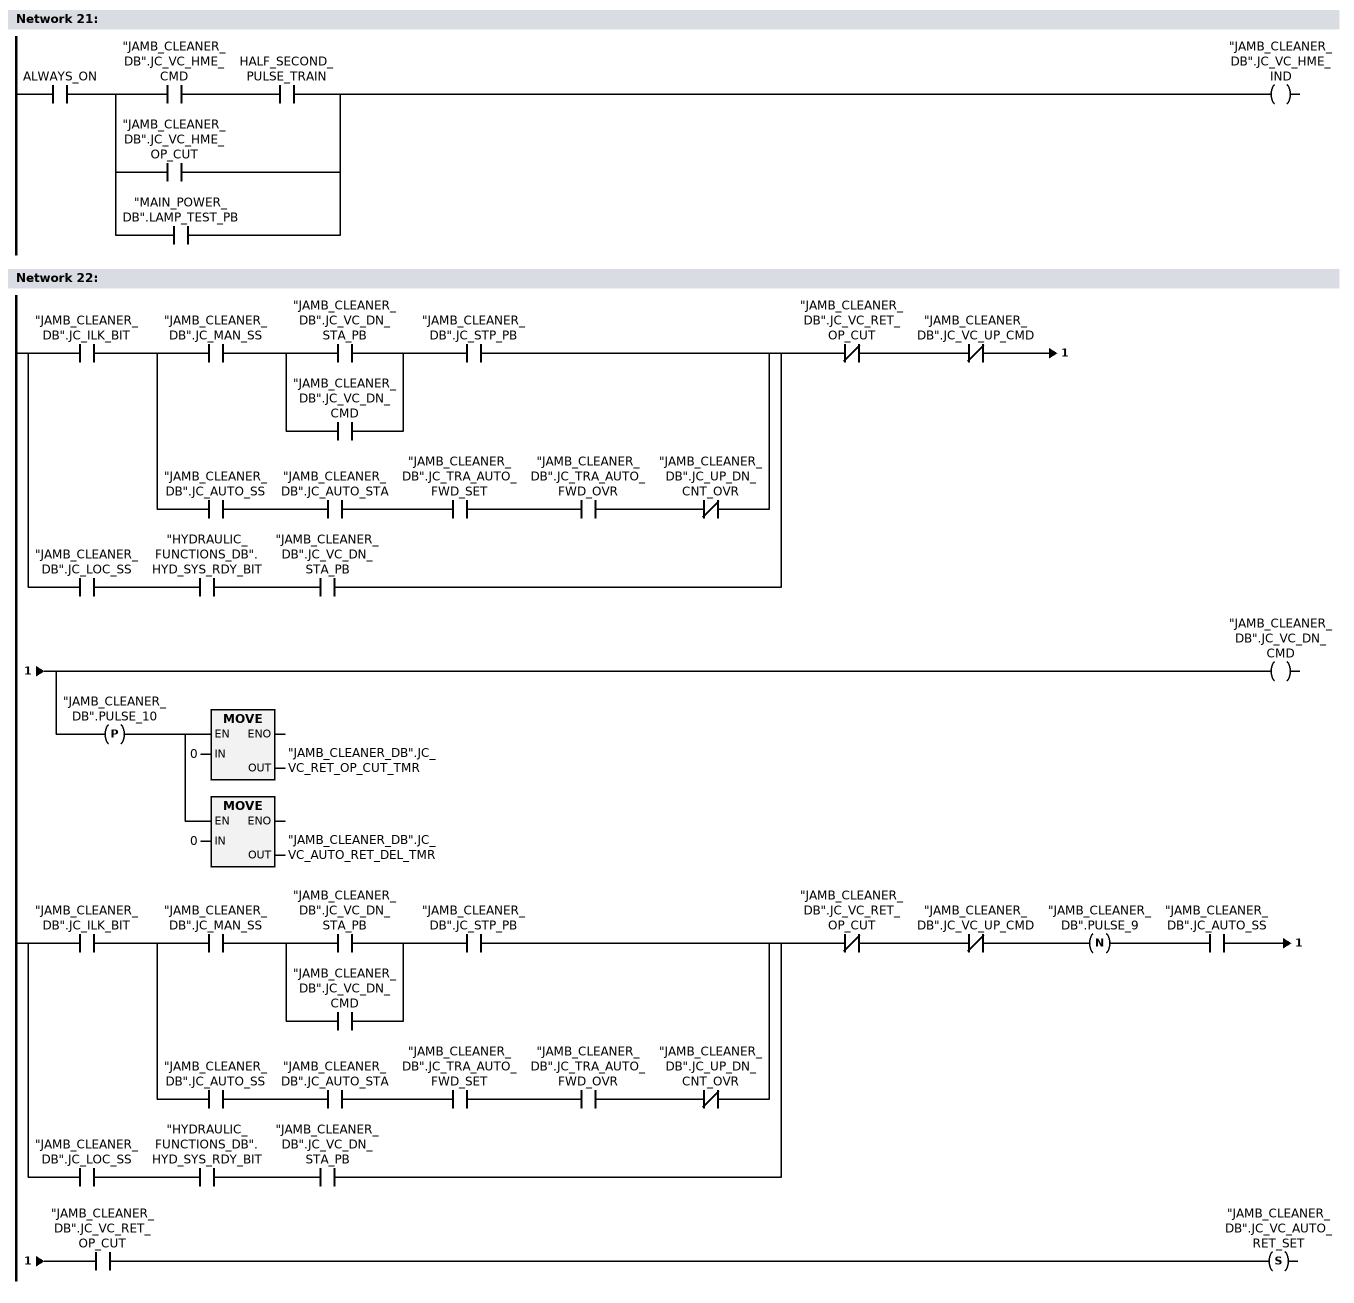
NETWORK
TITLE =
      A     "ALWAYS_ON";
      A(;
      A     "JAMB_CLEANER_DB".JC_VC_HME_CMD;
      A     "HALF_SECOND_PULSE_TRAIN";
      O     "JAMB_CLEANER_DB".JC_VC_HME_OP_CUT;
      O     "MAIN_POWER_DB".LAMP_TEST_PB;
      );
      =     "JAMB_CLEANER_DB".JC_VC_HME_IND;
NETWORK
TITLE =
      A(;
      A     "JAMB_CLEANER_DB".JC_ILK_BIT;
      A(;
      A     "JAMB_CLEANER_DB".JC_MAN_SS;
      A(;
      O     "JAMB_CLEANER_DB".JC_VC_DN_STA_PB;
      O     "JAMB_CLEANER_DB".JC_VC_DN_CMD;
      );
      A     "JAMB_CLEANER_DB".JC_STP_PB;
      O;
      A     "JAMB_CLEANER_DB".JC_AUTO_SS;
      A     "JAMB_CLEANER_DB".JC_AUTO_STA;
      A     "JAMB_CLEANER_DB".JC_TRA_AUTO_FWD_SET;
      A     "JAMB_CLEANER_DB".JC_TRA_AUTO_FWD_OVR;
      AN    "JAMB_CLEANER_DB".JC_UP_DN_CNT_OVR;
      );
      O;
      A     "JAMB_CLEANER_DB".JC_LOC_SS;
      A     "HYDRAULIC_FUNCTIONS_DB".HYD_SYS_RDY_BIT;
      A     "JAMB_CLEANER_DB".JC_VC_DN_STA_PB;
      );
      AN    "JAMB_CLEANER_DB".JC_VC_RET_OP_CUT;
      AN    "JAMB_CLEANER_DB".JC_VC_UP_CMD;
      =     L 0.0;
      A     L 0.0;
      BLD   102;
      =     "JAMB_CLEANER_DB".JC_VC_DN_CMD;
      A(;
      A     L 0.0;
      FN    "JAMB_CLEANER_DB".PULSE_9;
      );
      A     "JAMB_CLEANER_DB".JC_AUTO_SS;
      A     "JAMB_CLEANER_DB".JC_VC_RET_OP_CUT;
      S     "JAMB_CLEANER_DB".JC_VC_AUTO_RET_SET;
      A     L 0.0;
      FP    "JAMB_CLEANER_DB".PULSE_10;
      =     L 0.1;
      A     L 0.1;
      JNB   M018;
      L     0;
      T     "JAMB_CLEANER_DB".JC_VC_RET_OP_CUT_TMR;
M018: NOP   0;
      A     L 0.1;
      JNB   M019;
      L     0;
      T     "JAMB_CLEANER_DB".JC_VC_AUTO_RET_DEL_TMR;
M019: NOP   0;
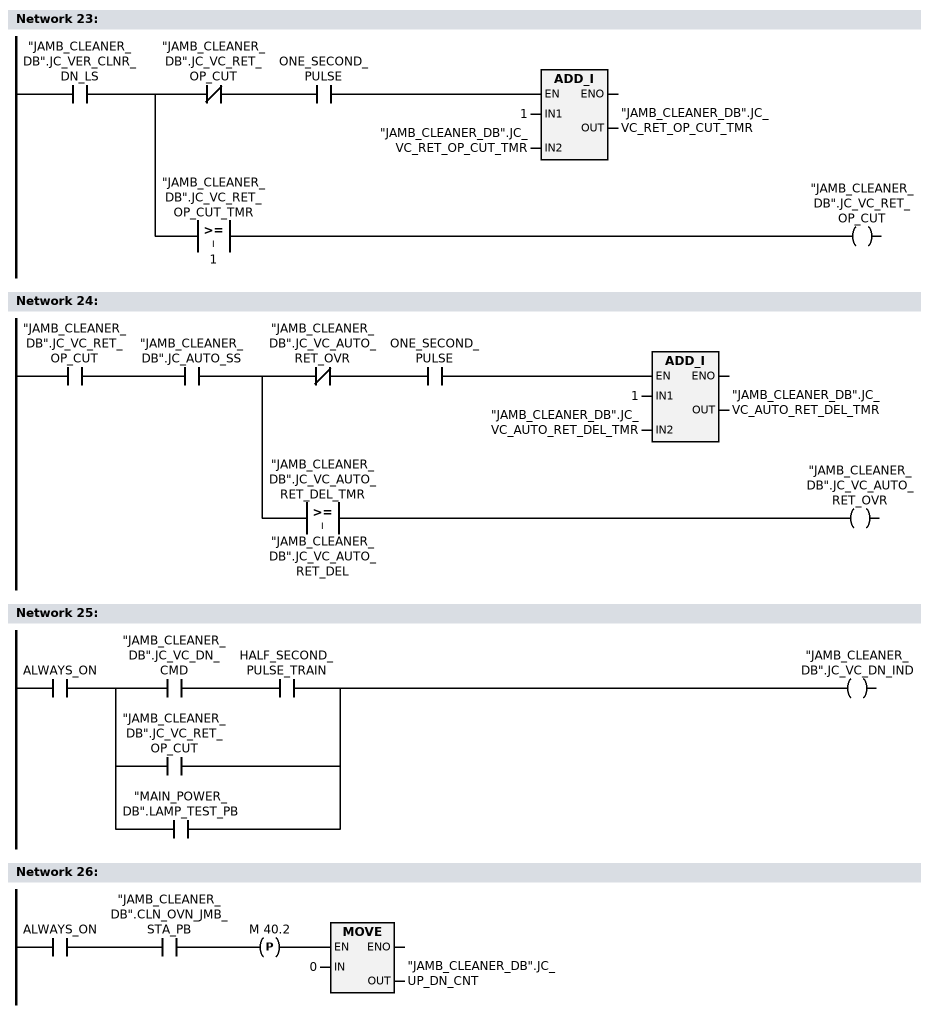
NETWORK
TITLE =
      A     "JAMB_CLEANER_DB".JC_VER_CLNR_DN_LS;
      =     L 0.0;
      A     L 0.0;
      AN    "JAMB_CLEANER_DB".JC_VC_RET_OP_CUT;
      A     "ONE_SECOND_PULSE";
      JNB   M020;
      L     1;
      L     "JAMB_CLEANER_DB".JC_VC_RET_OP_CUT_TMR;
      +I;
      T     "JAMB_CLEANER_DB".JC_VC_RET_OP_CUT_TMR;
M020: NOP   0;
      A     L 0.0;
      A(;
      L     "JAMB_CLEANER_DB".JC_VC_RET_OP_CUT_TMR;
      L     1;
      >=I;
      );
      =     "JAMB_CLEANER_DB".JC_VC_RET_OP_CUT;
NETWORK
TITLE =
      A     "JAMB_CLEANER_DB".JC_VC_RET_OP_CUT;
      A     "JAMB_CLEANER_DB".JC_AUTO_SS;
      =     L 0.0;
      A     L 0.0;
      AN    "JAMB_CLEANER_DB".JC_VC_AUTO_RET_OVR;
      A     "ONE_SECOND_PULSE";
      JNB   M021;
      L     1;
      L     "JAMB_CLEANER_DB".JC_VC_AUTO_RET_DEL_TMR;
      +I;
      T     "JAMB_CLEANER_DB".JC_VC_AUTO_RET_DEL_TMR;
M021: NOP   0;
      A     L 0.0;
      A(;
      L     "JAMB_CLEANER_DB".JC_VC_AUTO_RET_DEL_TMR;
      L     "JAMB_CLEANER_DB".JC_VC_AUTO_RET_DEL;
      >=I;
      );
      =     "JAMB_CLEANER_DB".JC_VC_AUTO_RET_OVR;
NETWORK
TITLE =
      A     "ALWAYS_ON";
      A(;
      A     "JAMB_CLEANER_DB".JC_VC_DN_CMD;
      A     "HALF_SECOND_PULSE_TRAIN";
      O     "JAMB_CLEANER_DB".JC_VC_RET_OP_CUT;
      O     "MAIN_POWER_DB".LAMP_TEST_PB;
      );
      =     "JAMB_CLEANER_DB".JC_VC_DN_IND;
NETWORK
TITLE =
      A     "ALWAYS_ON";
      A     "JAMB_CLEANER_DB".CLN_OVN_JMB_STA_PB;
      FP    M 40.2;
      JNB   M022;
      L     0;
      T     "JAMB_CLEANER_DB".JC_UP_DN_CNT;
M022: NOP   0;
END_FUNCTION

FUNCTION "GUIDE_CAGE" : VOID	// FC 11
AUTHOR : Kamillas
VERSION : 0.1
BEGIN
// (block stored without names or comments; labels and parameter names are numbered)
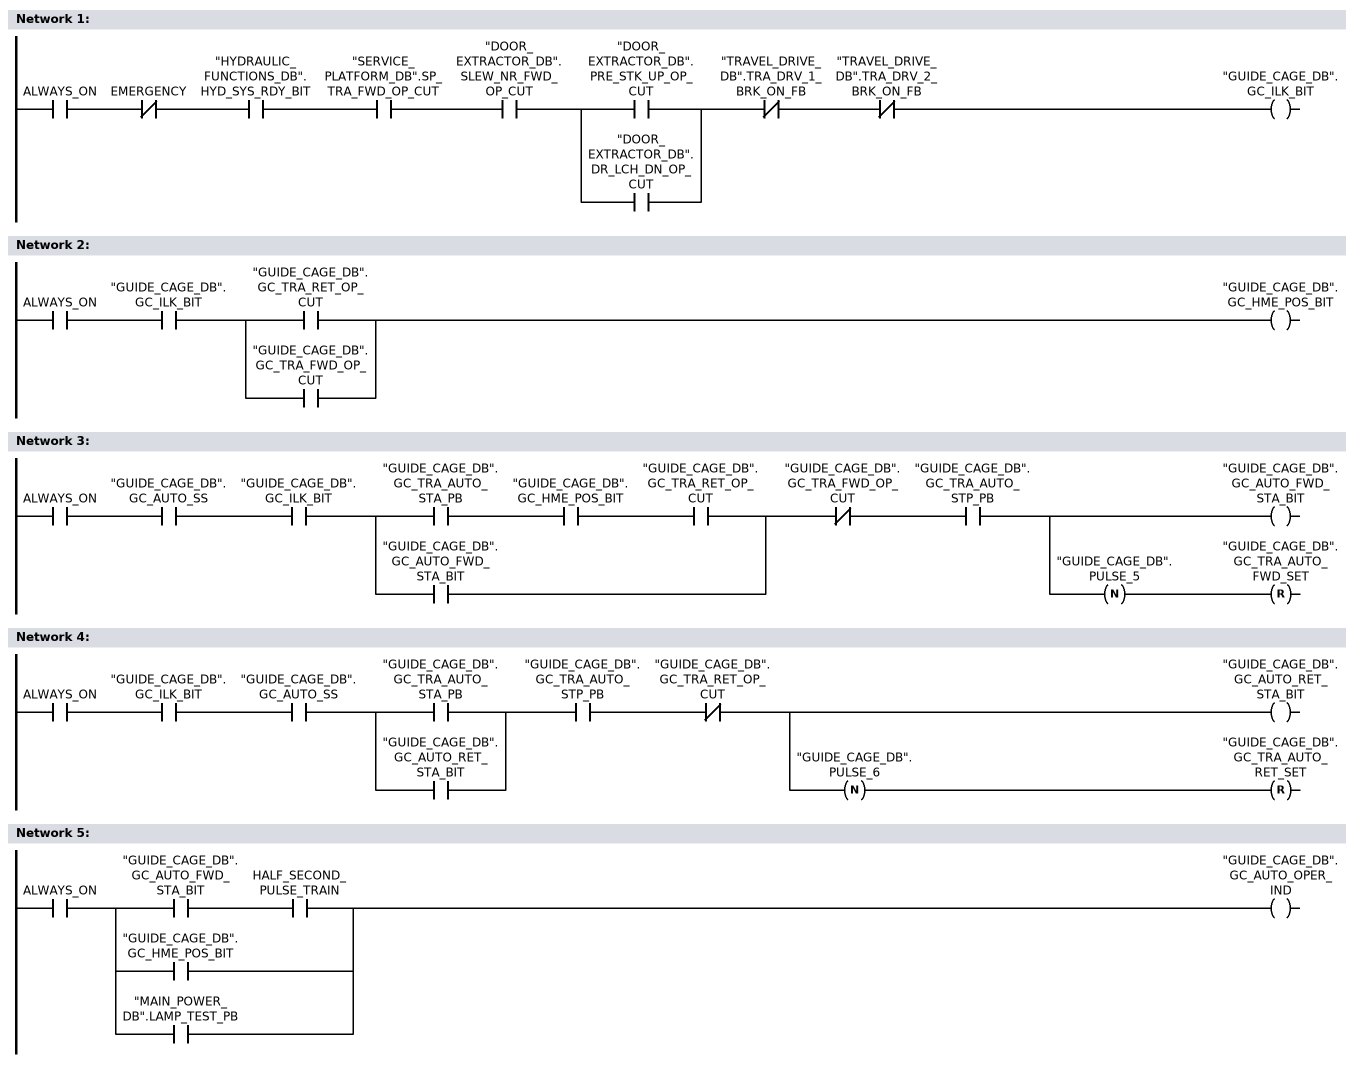
NETWORK
TITLE =
      A     "ALWAYS_ON";
      AN    "EMERGENCY";
      A     "HYDRAULIC_FUNCTIONS_DB".HYD_SYS_RDY_BIT;
      A     "SERVICE_PLATFORM_DB".SP_TRA_FWD_OP_CUT;
      A     "DOOR_EXTRACTOR_DB".SLEW_NR_FWD_OP_CUT;
      A(;
      O     "DOOR_EXTRACTOR_DB".PRE_STK_UP_OP_CUT;
      O     "DOOR_EXTRACTOR_DB".DR_LCH_DN_OP_CUT;
      );
      AN    "TRAVEL_DRIVE_DB".TRA_DRV_1_BRK_ON_FB;
      AN    "TRAVEL_DRIVE_DB".TRA_DRV_2_BRK_ON_FB;
      =     "GUIDE_CAGE_DB".GC_ILK_BIT;
NETWORK
TITLE =
      A     "ALWAYS_ON";
      A     "GUIDE_CAGE_DB".GC_ILK_BIT;
      A(;
      O     "GUIDE_CAGE_DB".GC_TRA_RET_OP_CUT;
      O     "GUIDE_CAGE_DB".GC_TRA_FWD_OP_CUT;
      );
      =     "GUIDE_CAGE_DB".GC_HME_POS_BIT;
NETWORK
TITLE =
      A     "ALWAYS_ON";
      A     "GUIDE_CAGE_DB".GC_AUTO_SS;
      A     "GUIDE_CAGE_DB".GC_ILK_BIT;
      A(;
      A     "GUIDE_CAGE_DB".GC_TRA_AUTO_STA_PB;
      A     "GUIDE_CAGE_DB".GC_HME_POS_BIT;
      A     "GUIDE_CAGE_DB".GC_TRA_RET_OP_CUT;
      O     "GUIDE_CAGE_DB".GC_AUTO_FWD_STA_BIT;
      );
      AN    "GUIDE_CAGE_DB".GC_TRA_FWD_OP_CUT;
      A     "GUIDE_CAGE_DB".GC_TRA_AUTO_STP_PB;
      =     L 0.0;
      A     L 0.0;
      BLD   102;
      =     "GUIDE_CAGE_DB".GC_AUTO_FWD_STA_BIT;
      A     L 0.0;
      FN    "GUIDE_CAGE_DB".PULSE_5;
      R     "GUIDE_CAGE_DB".GC_TRA_AUTO_FWD_SET;
NETWORK
TITLE =
      A     "ALWAYS_ON";
      A     "GUIDE_CAGE_DB".GC_ILK_BIT;
      A     "GUIDE_CAGE_DB".GC_AUTO_SS;
      A(;
      O     "GUIDE_CAGE_DB".GC_TRA_AUTO_STA_PB;
      O     "GUIDE_CAGE_DB".GC_AUTO_RET_STA_BIT;
      );
      A     "GUIDE_CAGE_DB".GC_TRA_AUTO_STP_PB;
      AN    "GUIDE_CAGE_DB".GC_TRA_RET_OP_CUT;
      =     L 0.0;
      A     L 0.0;
      BLD   102;
      =     "GUIDE_CAGE_DB".GC_AUTO_RET_STA_BIT;
      A     L 0.0;
      FN    "GUIDE_CAGE_DB".PULSE_6;
      R     "GUIDE_CAGE_DB".GC_TRA_AUTO_RET_SET;
NETWORK
TITLE =
      A     "ALWAYS_ON";
      A(;
      A     "GUIDE_CAGE_DB".GC_AUTO_FWD_STA_BIT;
      A     "HALF_SECOND_PULSE_TRAIN";
      O     "GUIDE_CAGE_DB".GC_HME_POS_BIT;
      O     "MAIN_POWER_DB".LAMP_TEST_PB;
      );
      =     "GUIDE_CAGE_DB".GC_AUTO_OPER_IND;
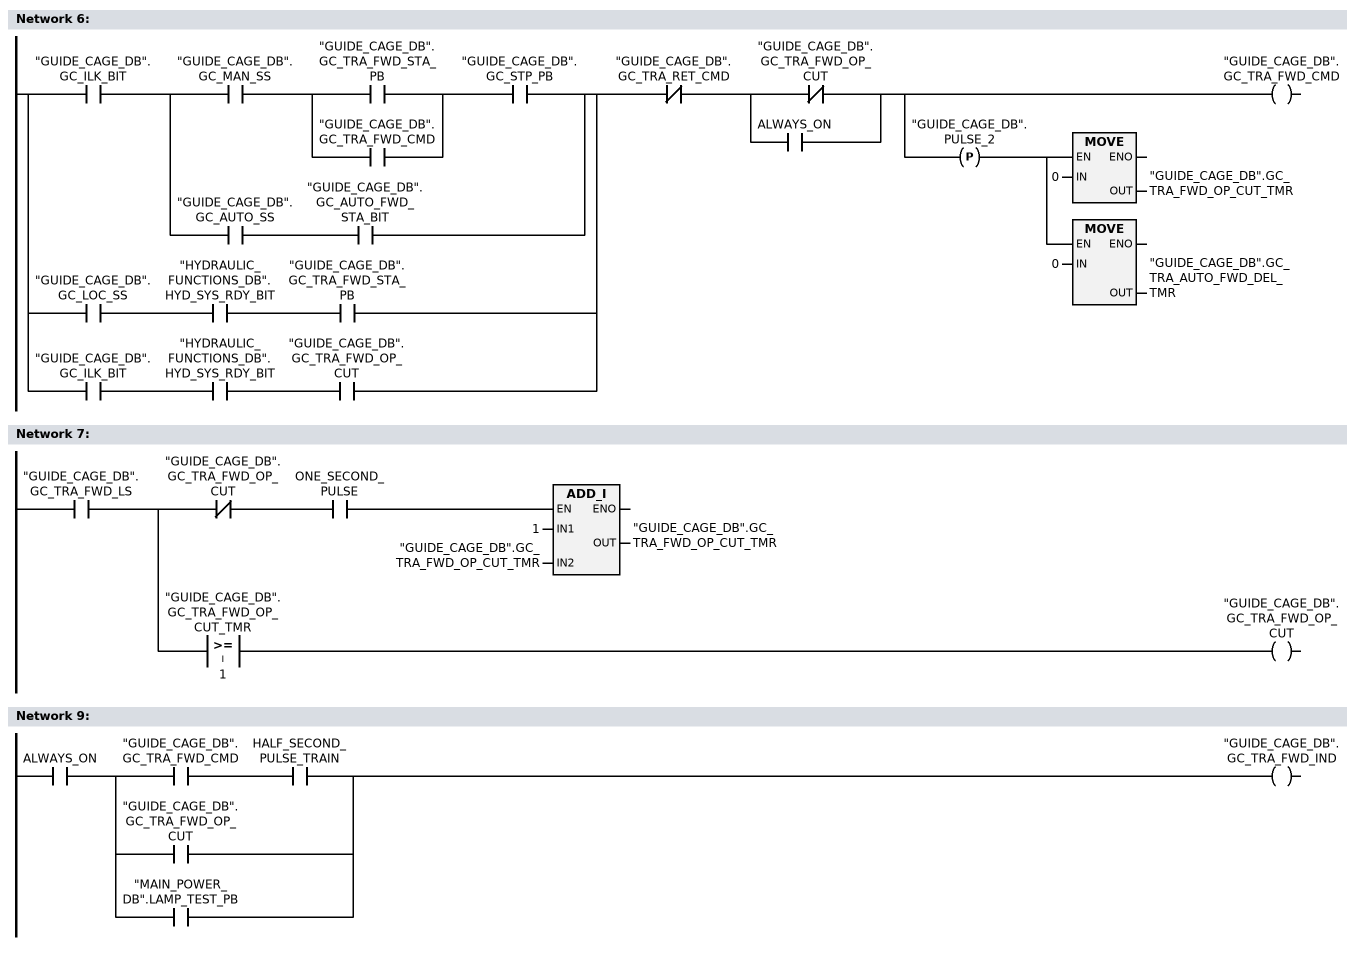
NETWORK
TITLE =
      A(;
      A     "GUIDE_CAGE_DB".GC_ILK_BIT;
      A(;
      A     "GUIDE_CAGE_DB".GC_MAN_SS;
      A(;
      O     "GUIDE_CAGE_DB".GC_TRA_FWD_STA_PB;
      O     "GUIDE_CAGE_DB".GC_TRA_FWD_CMD;
      );
      A     "GUIDE_CAGE_DB".GC_STP_PB;
      O;
      A     "GUIDE_CAGE_DB".GC_AUTO_SS;
      A     "GUIDE_CAGE_DB".GC_AUTO_FWD_STA_BIT;
      );
      O;
      A     "GUIDE_CAGE_DB".GC_LOC_SS;
      A     "HYDRAULIC_FUNCTIONS_DB".HYD_SYS_RDY_BIT;
      A     "GUIDE_CAGE_DB".GC_TRA_FWD_STA_PB;
      O;
      A     "GUIDE_CAGE_DB".GC_ILK_BIT;
      A     "HYDRAULIC_FUNCTIONS_DB".HYD_SYS_RDY_BIT;
      A     "GUIDE_CAGE_DB".GC_TRA_FWD_OP_CUT;
      );
      AN    "GUIDE_CAGE_DB".GC_TRA_RET_CMD;
      A(;
      ON    "GUIDE_CAGE_DB".GC_TRA_FWD_OP_CUT;
      O     "ALWAYS_ON";
      );
      =     L 0.0;
      A     L 0.0;
      BLD   102;
      =     "GUIDE_CAGE_DB".GC_TRA_FWD_CMD;
      A     L 0.0;
      FP    "GUIDE_CAGE_DB".PULSE_2;
      =     L 0.1;
      A     L 0.1;
      JNB   M001;
      L     0;
      T     "GUIDE_CAGE_DB".GC_TRA_FWD_OP_CUT_TMR;
M001: NOP   0;
      A     L 0.1;
      JNB   M002;
      L     0;
      T     "GUIDE_CAGE_DB".GC_TRA_AUTO_FWD_DEL_TMR;
M002: NOP   0;
NETWORK
TITLE =
      A     "GUIDE_CAGE_DB".GC_TRA_FWD_LS;
      =     L 0.0;
      A     L 0.0;
      AN    "GUIDE_CAGE_DB".GC_TRA_FWD_OP_CUT;
      A     "ONE_SECOND_PULSE";
      JNB   M003;
      L     1;
      L     "GUIDE_CAGE_DB".GC_TRA_FWD_OP_CUT_TMR;
      +I;
      T     "GUIDE_CAGE_DB".GC_TRA_FWD_OP_CUT_TMR;
M003: NOP   0;
      A     L 0.0;
      A(;
      L     "GUIDE_CAGE_DB".GC_TRA_FWD_OP_CUT_TMR;
      L     1;
      >=I;
      );
      =     "GUIDE_CAGE_DB".GC_TRA_FWD_OP_CUT;
NETWORK
TITLE =
      A     "GUIDE_CAGE_DB".GC_TRA_FWD_OP_CUT;
      =     L 0.0;
      A     L 0.0;
      A     "GUIDE_CAGE_DB".GC_AUTO_SS;
      AN    "GUIDE_CAGE_DB".GC_TRA_AUTO_FWD_OVR;
      A     "ONE_SECOND_PULSE";
      JNB   M004;
      L     1;
      L     "GUIDE_CAGE_DB".GC_TRA_AUTO_FWD_DEL_TMR;
      +I;
      T     "GUIDE_CAGE_DB".GC_TRA_AUTO_FWD_DEL_TMR;
M004: NOP   0;
      A     L 0.0;
      A(;
      L     "GUIDE_CAGE_DB".GC_TRA_AUTO_FWD_DEL_TMR;
      L     "GUIDE_CAGE_DB".GC_TRA_AUTO_FWD_DEL;
      >=I;
      );
      =     L 0.1;
      A     L 0.1;
      A     "GUIDE_CAGE_DB".GC_AUTO_SS;
      =     "GUIDE_CAGE_DB".GC_TRA_AUTO_FWD_OVR;
      A(;
      A     L 0.1;
      FP    "GUIDE_CAGE_DB".PULSE_1;
      );
      A     "GUIDE_CAGE_DB".GC_AUTO_SS;
      A     "GUIDE_CAGE_DB".GC_TRA_FWD_OP_CUT;
      S     "GUIDE_CAGE_DB".GC_TRA_AUTO_FWD_SET;
NETWORK
TITLE =
      A     "ALWAYS_ON";
      A(;
      A     "GUIDE_CAGE_DB".GC_TRA_FWD_CMD;
      A     "HALF_SECOND_PULSE_TRAIN";
      O     "GUIDE_CAGE_DB".GC_TRA_FWD_OP_CUT;
      O     "MAIN_POWER_DB".LAMP_TEST_PB;
      );
      =     "GUIDE_CAGE_DB".GC_TRA_FWD_IND;
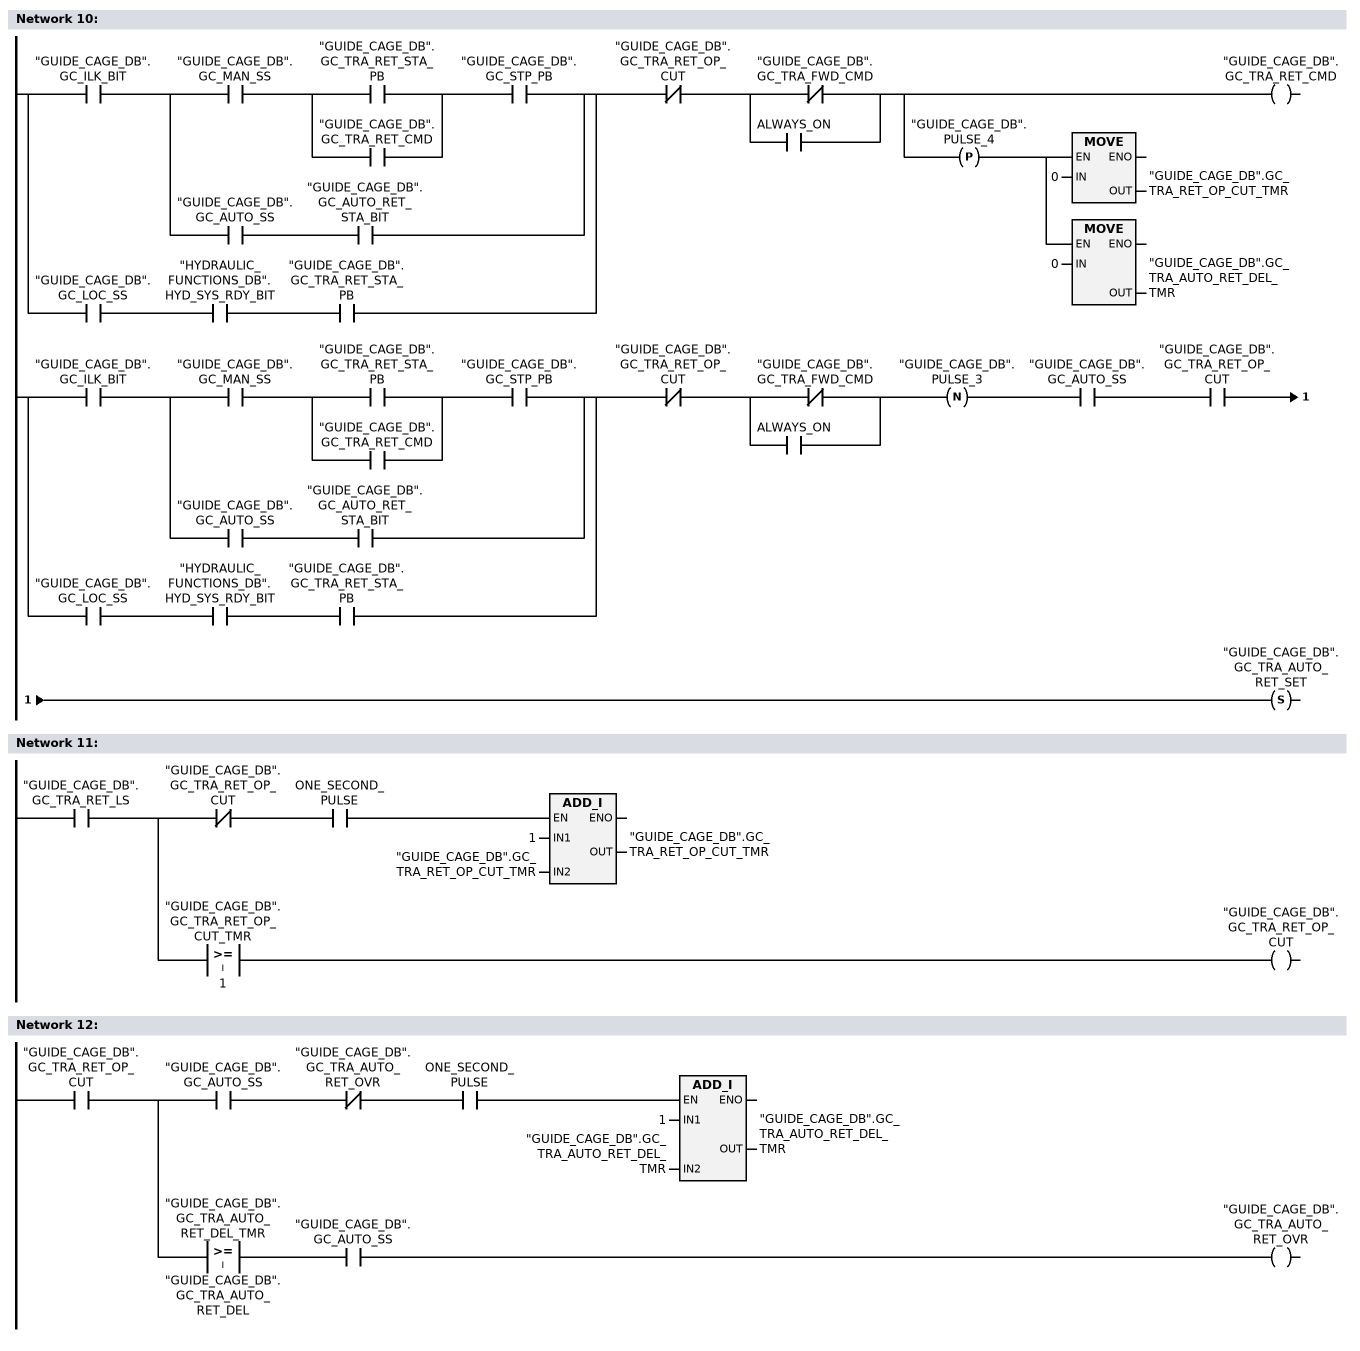
NETWORK
TITLE =
      A(;
      A     "GUIDE_CAGE_DB".GC_ILK_BIT;
      A(;
      A     "GUIDE_CAGE_DB".GC_MAN_SS;
      A(;
      O     "GUIDE_CAGE_DB".GC_TRA_RET_STA_PB;
      O     "GUIDE_CAGE_DB".GC_TRA_RET_CMD;
      );
      A     "GUIDE_CAGE_DB".GC_STP_PB;
      O;
      A     "GUIDE_CAGE_DB".GC_AUTO_SS;
      A     "GUIDE_CAGE_DB".GC_AUTO_RET_STA_BIT;
      );
      O;
      A     "GUIDE_CAGE_DB".GC_LOC_SS;
      A     "HYDRAULIC_FUNCTIONS_DB".HYD_SYS_RDY_BIT;
      A     "GUIDE_CAGE_DB".GC_TRA_RET_STA_PB;
      );
      AN    "GUIDE_CAGE_DB".GC_TRA_RET_OP_CUT;
      A(;
      ON    "GUIDE_CAGE_DB".GC_TRA_FWD_CMD;
      O     "ALWAYS_ON";
      );
      =     L 0.0;
      A     L 0.0;
      BLD   102;
      =     "GUIDE_CAGE_DB".GC_TRA_RET_CMD;
      A(;
      A     L 0.0;
      FN    "GUIDE_CAGE_DB".PULSE_3;
      );
      A     "GUIDE_CAGE_DB".GC_AUTO_SS;
      A     "GUIDE_CAGE_DB".GC_TRA_RET_OP_CUT;
      S     "GUIDE_CAGE_DB".GC_TRA_AUTO_RET_SET;
      A     L 0.0;
      FP    "GUIDE_CAGE_DB".PULSE_4;
      =     L 0.1;
      A     L 0.1;
      JNB   M005;
      L     0;
      T     "GUIDE_CAGE_DB".GC_TRA_RET_OP_CUT_TMR;
M005: NOP   0;
      A     L 0.1;
      JNB   M006;
      L     0;
      T     "GUIDE_CAGE_DB".GC_TRA_AUTO_RET_DEL_TMR;
M006: NOP   0;
NETWORK
TITLE =
      A     "GUIDE_CAGE_DB".GC_TRA_RET_LS;
      =     L 0.0;
      A     L 0.0;
      AN    "GUIDE_CAGE_DB".GC_TRA_RET_OP_CUT;
      A     "ONE_SECOND_PULSE";
      JNB   M007;
      L     1;
      L     "GUIDE_CAGE_DB".GC_TRA_RET_OP_CUT_TMR;
      +I;
      T     "GUIDE_CAGE_DB".GC_TRA_RET_OP_CUT_TMR;
M007: NOP   0;
      A     L 0.0;
      A(;
      L     "GUIDE_CAGE_DB".GC_TRA_RET_OP_CUT_TMR;
      L     1;
      >=I;
      );
      =     "GUIDE_CAGE_DB".GC_TRA_RET_OP_CUT;
NETWORK
TITLE =
      A     "GUIDE_CAGE_DB".GC_TRA_RET_OP_CUT;
      =     L 0.0;
      A     L 0.0;
      A     "GUIDE_CAGE_DB".GC_AUTO_SS;
      AN    "GUIDE_CAGE_DB".GC_TRA_AUTO_RET_OVR;
      A     "ONE_SECOND_PULSE";
      JNB   M008;
      L     1;
      L     "GUIDE_CAGE_DB".GC_TRA_AUTO_RET_DEL_TMR;
      +I;
      T     "GUIDE_CAGE_DB".GC_TRA_AUTO_RET_DEL_TMR;
M008: NOP   0;
      A     L 0.0;
      A(;
      L     "GUIDE_CAGE_DB".GC_TRA_AUTO_RET_DEL_TMR;
      L     "GUIDE_CAGE_DB".GC_TRA_AUTO_RET_DEL;
      >=I;
      );
      A     "GUIDE_CAGE_DB".GC_AUTO_SS;
      =     "GUIDE_CAGE_DB".GC_TRA_AUTO_RET_OVR;
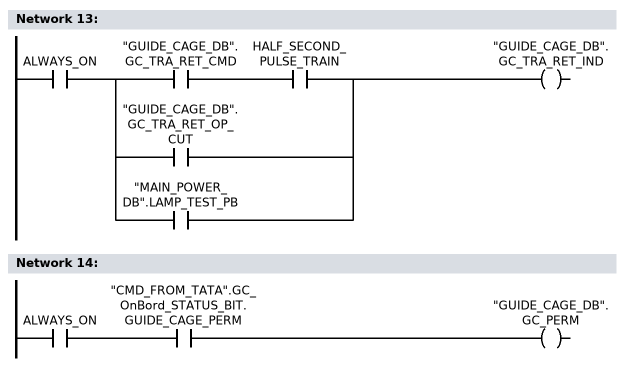
NETWORK
TITLE =
      A     "ALWAYS_ON";
      A(;
      A     "GUIDE_CAGE_DB".GC_TRA_RET_CMD;
      A     "HALF_SECOND_PULSE_TRAIN";
      O     "GUIDE_CAGE_DB".GC_TRA_RET_OP_CUT;
      O     "MAIN_POWER_DB".LAMP_TEST_PB;
      );
      =     "GUIDE_CAGE_DB".GC_TRA_RET_IND;
NETWORK
TITLE =
      A     "ALWAYS_ON";
      A     "CMD_FROM_TATA".GC_OnBord_STATUS_BIT.GUIDE_CAGE_PERM;
      =     "GUIDE_CAGE_DB".GC_PERM;
END_FUNCTION

FUNCTION "DOOR_CLEANER_MOTOR" : VOID	// FC 12
AUTHOR : Kamillas
VERSION : 0.1
BEGIN
// (block stored without names or comments; labels and parameter names are numbered)
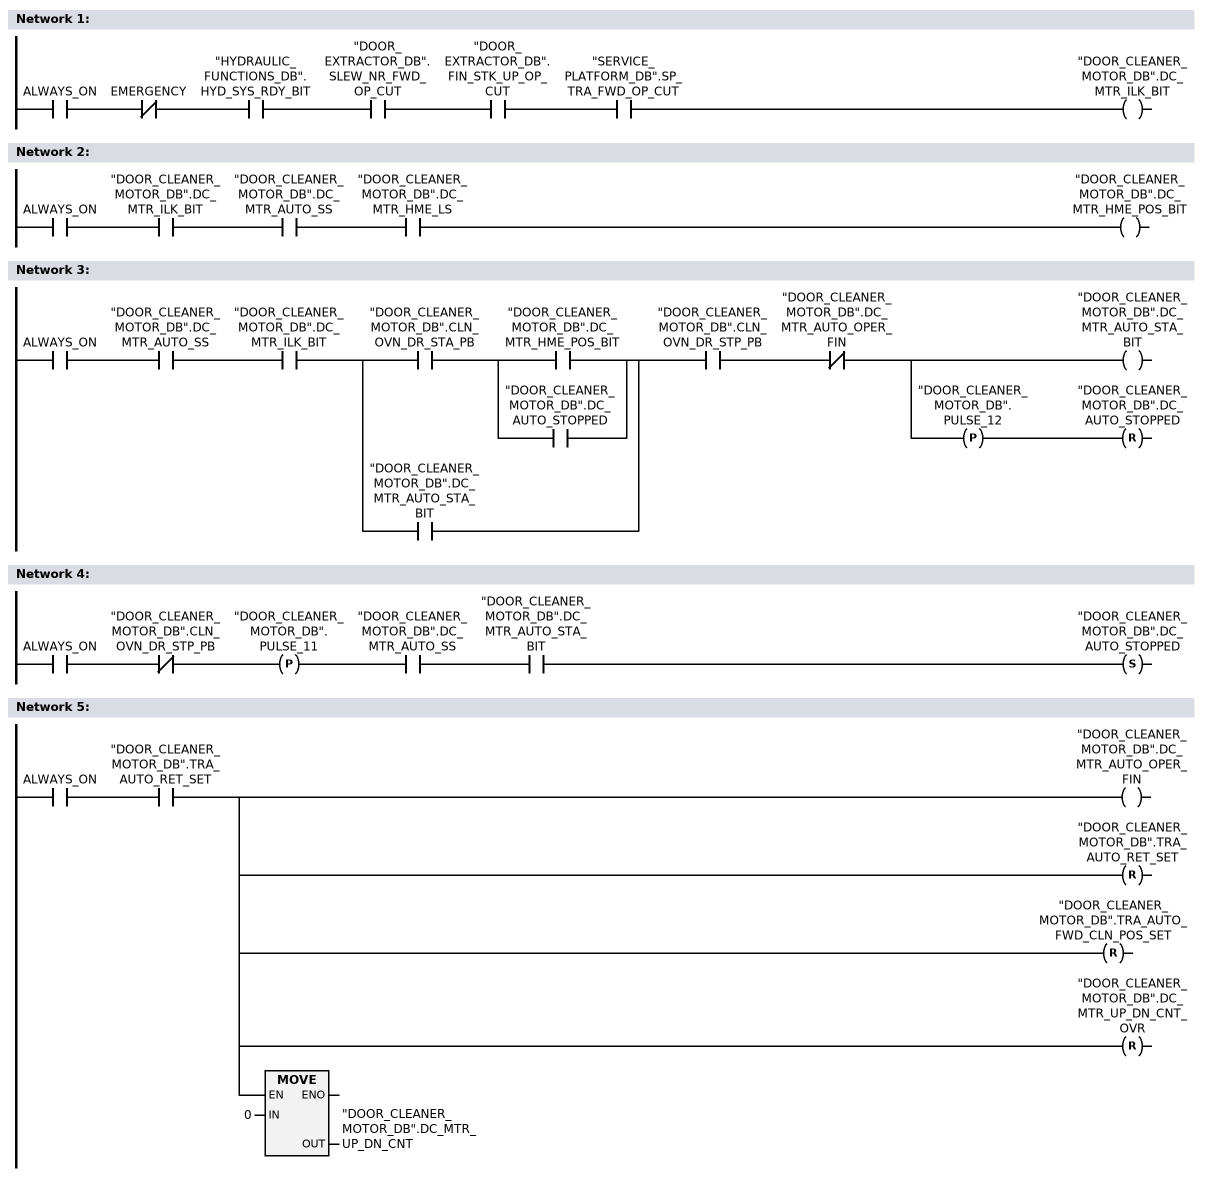
NETWORK
TITLE =
      A     "ALWAYS_ON";
      AN    "EMERGENCY";
      A     "HYDRAULIC_FUNCTIONS_DB".HYD_SYS_RDY_BIT;
      A     "DOOR_EXTRACTOR_DB".SLEW_NR_FWD_OP_CUT;
      A     "DOOR_EXTRACTOR_DB".FIN_STK_UP_OP_CUT;
      A     "SERVICE_PLATFORM_DB".SP_TRA_FWD_OP_CUT;
      =     "DOOR_CLEANER_MOTOR_DB".DC_MTR_ILK_BIT;
NETWORK
TITLE =
      A     "ALWAYS_ON";
      A     "DOOR_CLEANER_MOTOR_DB".DC_MTR_ILK_BIT;
      A     "DOOR_CLEANER_MOTOR_DB".DC_MTR_AUTO_SS;
      A     "DOOR_CLEANER_MOTOR_DB".DC_MTR_HME_LS;
      =     "DOOR_CLEANER_MOTOR_DB".DC_MTR_HME_POS_BIT;
NETWORK
TITLE =
      A     "ALWAYS_ON";
      A     "DOOR_CLEANER_MOTOR_DB".DC_MTR_AUTO_SS;
      A     "DOOR_CLEANER_MOTOR_DB".DC_MTR_ILK_BIT;
      A(;
      A     "DOOR_CLEANER_MOTOR_DB".CLN_OVN_DR_STA_PB;
      A(;
      O     "DOOR_CLEANER_MOTOR_DB".DC_MTR_HME_POS_BIT;
      O     "DOOR_CLEANER_MOTOR_DB".DC_AUTO_STOPPED;
      );
      O     "DOOR_CLEANER_MOTOR_DB".DC_MTR_AUTO_STA_BIT;
      );
      A     "DOOR_CLEANER_MOTOR_DB".CLN_OVN_DR_STP_PB;
      AN    "DOOR_CLEANER_MOTOR_DB".DC_MTR_AUTO_OPER_FIN;
      =     L 0.0;
      A     L 0.0;
      BLD   102;
      =     "DOOR_CLEANER_MOTOR_DB".DC_MTR_AUTO_STA_BIT;
      A     L 0.0;
      FP    "DOOR_CLEANER_MOTOR_DB".PULSE_12;
      R     "DOOR_CLEANER_MOTOR_DB".DC_AUTO_STOPPED;
NETWORK
TITLE =
      A     "ALWAYS_ON";
      AN    "DOOR_CLEANER_MOTOR_DB".CLN_OVN_DR_STP_PB;
      FP    "DOOR_CLEANER_MOTOR_DB".PULSE_11;
      A     "DOOR_CLEANER_MOTOR_DB".DC_MTR_AUTO_SS;
      A     "DOOR_CLEANER_MOTOR_DB".DC_MTR_AUTO_STA_BIT;
      S     "DOOR_CLEANER_MOTOR_DB".DC_AUTO_STOPPED;
NETWORK
TITLE =
      A     "ALWAYS_ON";
      A     "DOOR_CLEANER_MOTOR_DB".TRA_AUTO_RET_SET;
      =     L 0.0;
      A     L 0.0;
      BLD   102;
      =     "DOOR_CLEANER_MOTOR_DB".DC_MTR_AUTO_OPER_FIN;
      A     L 0.0;
      BLD   102;
      R     "DOOR_CLEANER_MOTOR_DB".TRA_AUTO_RET_SET;
      A     L 0.0;
      BLD   102;
      R     "DOOR_CLEANER_MOTOR_DB".TRA_AUTO_FWD_CLN_POS_SET;
      A     L 0.0;
      BLD   102;
      R     "DOOR_CLEANER_MOTOR_DB".DC_MTR_UP_DN_CNT_OVR;
      A     L 0.0;
      JNB   M001;
      L     0;
      T     "DOOR_CLEANER_MOTOR_DB".DC_MTR_UP_DN_CNT;
M001: NOP   0;
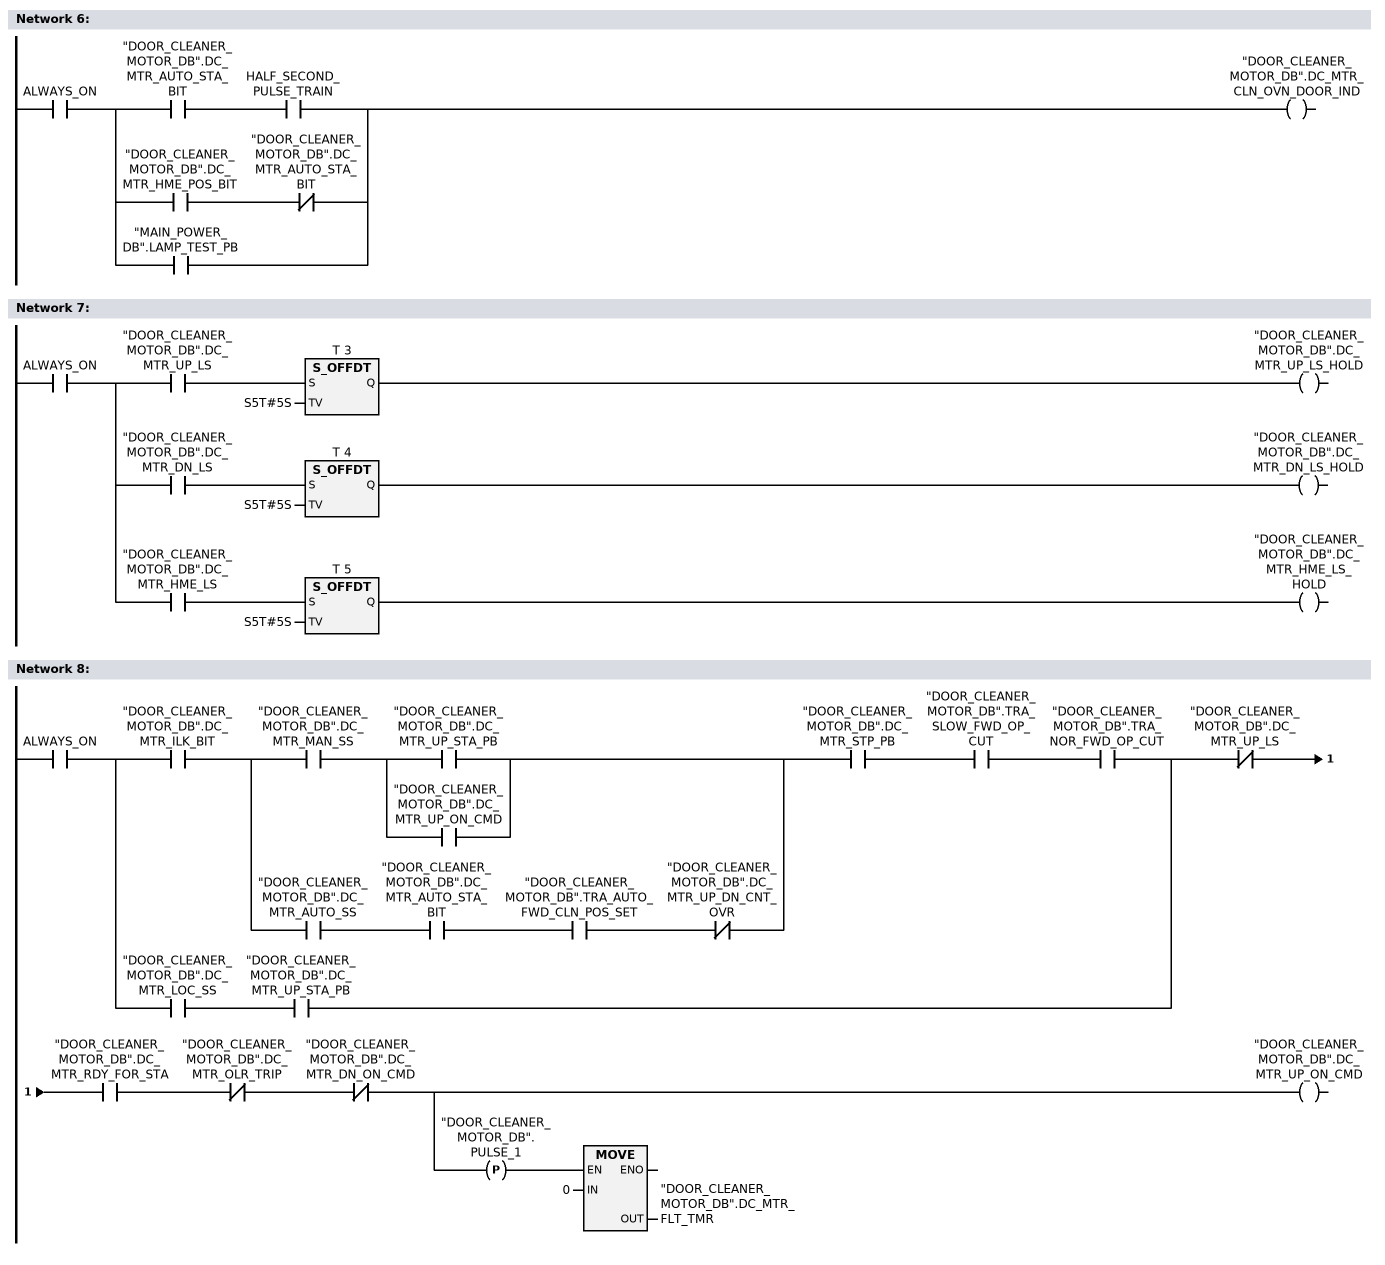
NETWORK
TITLE =
      A     "ALWAYS_ON";
      A(;
      A     "DOOR_CLEANER_MOTOR_DB".DC_MTR_AUTO_STA_BIT;
      A     "HALF_SECOND_PULSE_TRAIN";
      O;
      A     "DOOR_CLEANER_MOTOR_DB".DC_MTR_HME_POS_BIT;
      AN    "DOOR_CLEANER_MOTOR_DB".DC_MTR_AUTO_STA_BIT;
      O     "MAIN_POWER_DB".LAMP_TEST_PB;
      );
      =     "DOOR_CLEANER_MOTOR_DB".DC_MTR_CLN_OVN_DOOR_IND;
NETWORK
TITLE =
      A     "ALWAYS_ON";
      =     L 0.0;
      A     L 0.0;
      A     "DOOR_CLEANER_MOTOR_DB".DC_MTR_UP_LS;
      L     S5T#5S;
      SF    T 3;
      NOP   0;
      NOP   0;
      NOP   0;
      A     T 3;
      =     "DOOR_CLEANER_MOTOR_DB".DC_MTR_UP_LS_HOLD;
      A     L 0.0;
      A     "DOOR_CLEANER_MOTOR_DB".DC_MTR_DN_LS;
      L     S5T#5S;
      SF    T 4;
      NOP   0;
      NOP   0;
      NOP   0;
      A     T 4;
      =     "DOOR_CLEANER_MOTOR_DB".DC_MTR_DN_LS_HOLD;
      A     L 0.0;
      A     "DOOR_CLEANER_MOTOR_DB".DC_MTR_HME_LS;
      L     S5T#5S;
      SF    T 5;
      NOP   0;
      NOP   0;
      NOP   0;
      A     T 5;
      =     "DOOR_CLEANER_MOTOR_DB".DC_MTR_HME_LS_HOLD;
NETWORK
TITLE =
      A     "ALWAYS_ON";
      A(;
      A     "DOOR_CLEANER_MOTOR_DB".DC_MTR_ILK_BIT;
      A(;
      A     "DOOR_CLEANER_MOTOR_DB".DC_MTR_MAN_SS;
      A(;
      O     "DOOR_CLEANER_MOTOR_DB".DC_MTR_UP_STA_PB;
      O     "DOOR_CLEANER_MOTOR_DB".DC_MTR_UP_ON_CMD;
      );
      O;
      A     "DOOR_CLEANER_MOTOR_DB".DC_MTR_AUTO_SS;
      A     "DOOR_CLEANER_MOTOR_DB".DC_MTR_AUTO_STA_BIT;
      A     "DOOR_CLEANER_MOTOR_DB".TRA_AUTO_FWD_CLN_POS_SET;
      AN    "DOOR_CLEANER_MOTOR_DB".DC_MTR_UP_DN_CNT_OVR;
      );
      A     "DOOR_CLEANER_MOTOR_DB".DC_MTR_STP_PB;
      A     "DOOR_CLEANER_MOTOR_DB".TRA_SLOW_FWD_OP_CUT;
      A     "DOOR_CLEANER_MOTOR_DB".TRA_NOR_FWD_OP_CUT;
      O;
      A     "DOOR_CLEANER_MOTOR_DB".DC_MTR_LOC_SS;
      A     "DOOR_CLEANER_MOTOR_DB".DC_MTR_UP_STA_PB;
      );
      AN    "DOOR_CLEANER_MOTOR_DB".DC_MTR_UP_LS;
      A     "DOOR_CLEANER_MOTOR_DB".DC_MTR_RDY_FOR_STA;
      AN    "DOOR_CLEANER_MOTOR_DB".DC_MTR_OLR_TRIP;
      AN    "DOOR_CLEANER_MOTOR_DB".DC_MTR_DN_ON_CMD;
      =     L 0.0;
      A     L 0.0;
      BLD   102;
      =     "DOOR_CLEANER_MOTOR_DB".DC_MTR_UP_ON_CMD;
      A     L 0.0;
      FP    "DOOR_CLEANER_MOTOR_DB".PULSE_1;
      JNB   M002;
      L     0;
      T     "DOOR_CLEANER_MOTOR_DB".DC_MTR_FLT_TMR;
M002: NOP   0;
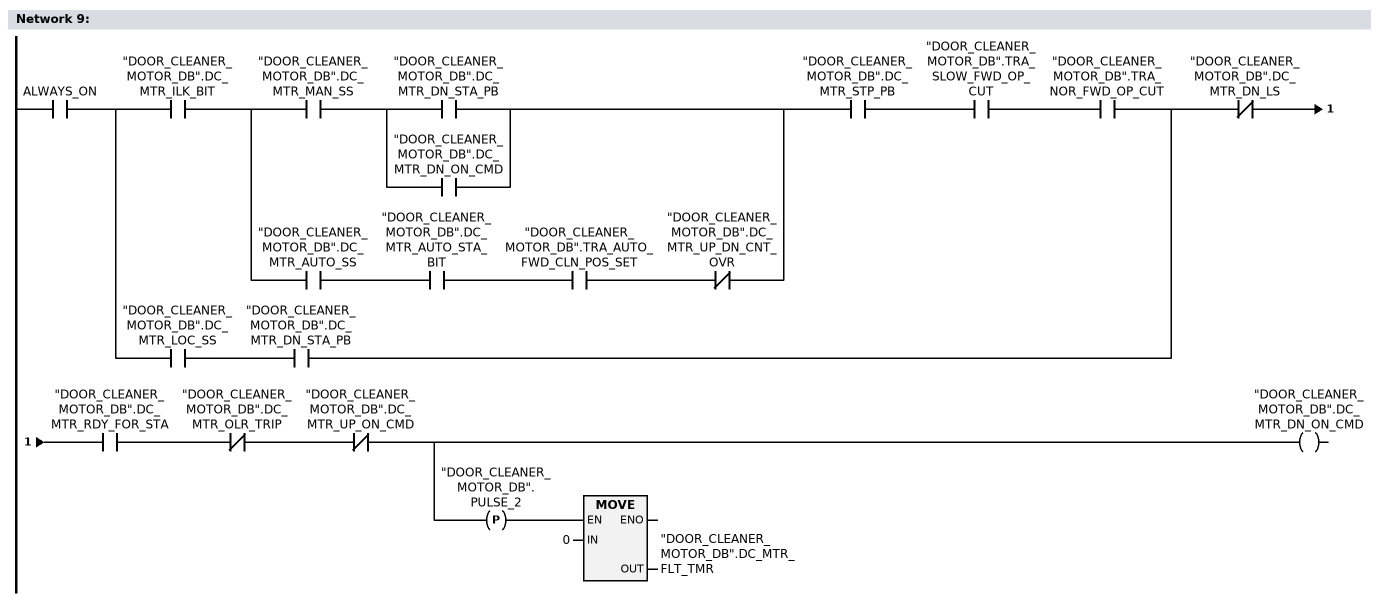
NETWORK
TITLE =
      A     "ALWAYS_ON";
      A(;
      A     "DOOR_CLEANER_MOTOR_DB".DC_MTR_ILK_BIT;
      A(;
      A     "DOOR_CLEANER_MOTOR_DB".DC_MTR_MAN_SS;
      A(;
      O     "DOOR_CLEANER_MOTOR_DB".DC_MTR_DN_STA_PB;
      O     "DOOR_CLEANER_MOTOR_DB".DC_MTR_DN_ON_CMD;
      );
      O;
      A     "DOOR_CLEANER_MOTOR_DB".DC_MTR_AUTO_SS;
      A     "DOOR_CLEANER_MOTOR_DB".DC_MTR_AUTO_STA_BIT;
      A     "DOOR_CLEANER_MOTOR_DB".TRA_AUTO_FWD_CLN_POS_SET;
      AN    "DOOR_CLEANER_MOTOR_DB".DC_MTR_UP_DN_CNT_OVR;
      );
      A     "DOOR_CLEANER_MOTOR_DB".DC_MTR_STP_PB;
      A     "DOOR_CLEANER_MOTOR_DB".TRA_SLOW_FWD_OP_CUT;
      A     "DOOR_CLEANER_MOTOR_DB".TRA_NOR_FWD_OP_CUT;
      O;
      A     "DOOR_CLEANER_MOTOR_DB".DC_MTR_LOC_SS;
      A     "DOOR_CLEANER_MOTOR_DB".DC_MTR_DN_STA_PB;
      );
      AN    "DOOR_CLEANER_MOTOR_DB".DC_MTR_DN_LS;
      A     "DOOR_CLEANER_MOTOR_DB".DC_MTR_RDY_FOR_STA;
      AN    "DOOR_CLEANER_MOTOR_DB".DC_MTR_OLR_TRIP;
      AN    "DOOR_CLEANER_MOTOR_DB".DC_MTR_UP_ON_CMD;
      =     L 0.0;
      A     L 0.0;
      BLD   102;
      =     "DOOR_CLEANER_MOTOR_DB".DC_MTR_DN_ON_CMD;
      A     L 0.0;
      FP    "DOOR_CLEANER_MOTOR_DB".PULSE_2;
      JNB   M003;
      L     0;
      T     "DOOR_CLEANER_MOTOR_DB".DC_MTR_FLT_TMR;
M003: NOP   0;
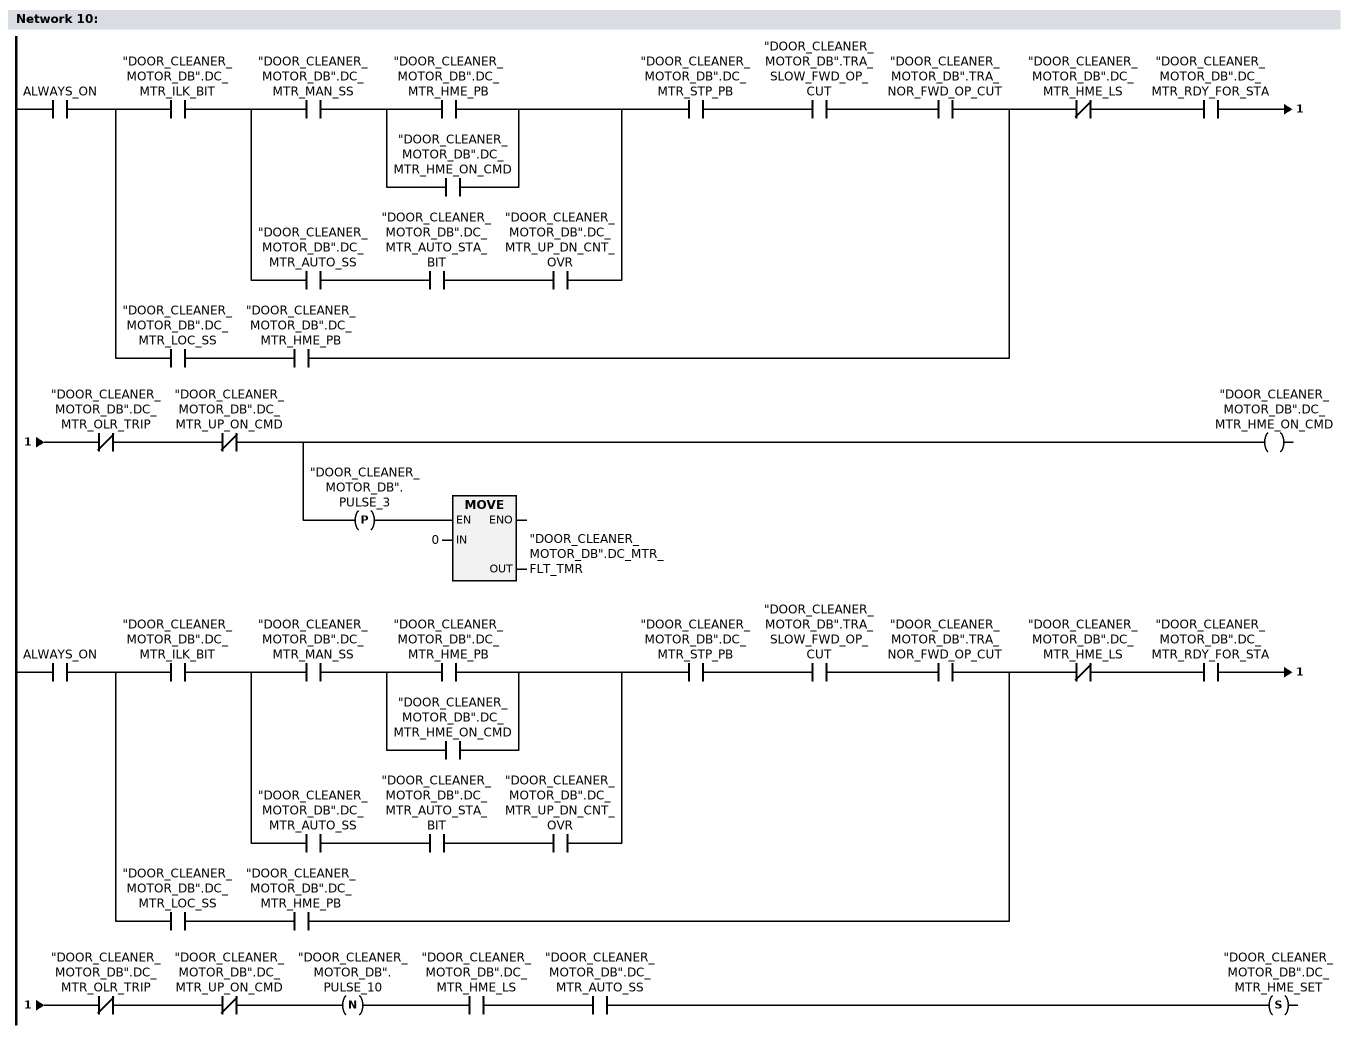
NETWORK
TITLE =
      A     "ALWAYS_ON";
      A(;
      A     "DOOR_CLEANER_MOTOR_DB".DC_MTR_ILK_BIT;
      A(;
      A     "DOOR_CLEANER_MOTOR_DB".DC_MTR_MAN_SS;
      A(;
      O     "DOOR_CLEANER_MOTOR_DB".DC_MTR_HME_PB;
      O     "DOOR_CLEANER_MOTOR_DB".DC_MTR_HME_ON_CMD;
      );
      O;
      A     "DOOR_CLEANER_MOTOR_DB".DC_MTR_AUTO_SS;
      A     "DOOR_CLEANER_MOTOR_DB".DC_MTR_AUTO_STA_BIT;
      A     "DOOR_CLEANER_MOTOR_DB".DC_MTR_UP_DN_CNT_OVR;
      );
      A     "DOOR_CLEANER_MOTOR_DB".DC_MTR_STP_PB;
      A     "DOOR_CLEANER_MOTOR_DB".TRA_SLOW_FWD_OP_CUT;
      A     "DOOR_CLEANER_MOTOR_DB".TRA_NOR_FWD_OP_CUT;
      O;
      A     "DOOR_CLEANER_MOTOR_DB".DC_MTR_LOC_SS;
      A     "DOOR_CLEANER_MOTOR_DB".DC_MTR_HME_PB;
      );
      AN    "DOOR_CLEANER_MOTOR_DB".DC_MTR_HME_LS;
      A     "DOOR_CLEANER_MOTOR_DB".DC_MTR_RDY_FOR_STA;
      AN    "DOOR_CLEANER_MOTOR_DB".DC_MTR_OLR_TRIP;
      AN    "DOOR_CLEANER_MOTOR_DB".DC_MTR_UP_ON_CMD;
      =     L 0.0;
      A     L 0.0;
      BLD   102;
      =     "DOOR_CLEANER_MOTOR_DB".DC_MTR_HME_ON_CMD;
      A(;
      A     L 0.0;
      FN    "DOOR_CLEANER_MOTOR_DB".PULSE_10;
      );
      A     "DOOR_CLEANER_MOTOR_DB".DC_MTR_HME_LS;
      A     "DOOR_CLEANER_MOTOR_DB".DC_MTR_AUTO_SS;
      S     "DOOR_CLEANER_MOTOR_DB".DC_MTR_HME_SET;
      A     L 0.0;
      FP    "DOOR_CLEANER_MOTOR_DB".PULSE_3;
      JNB   M004;
      L     0;
      T     "DOOR_CLEANER_MOTOR_DB".DC_MTR_FLT_TMR;
M004: NOP   0;
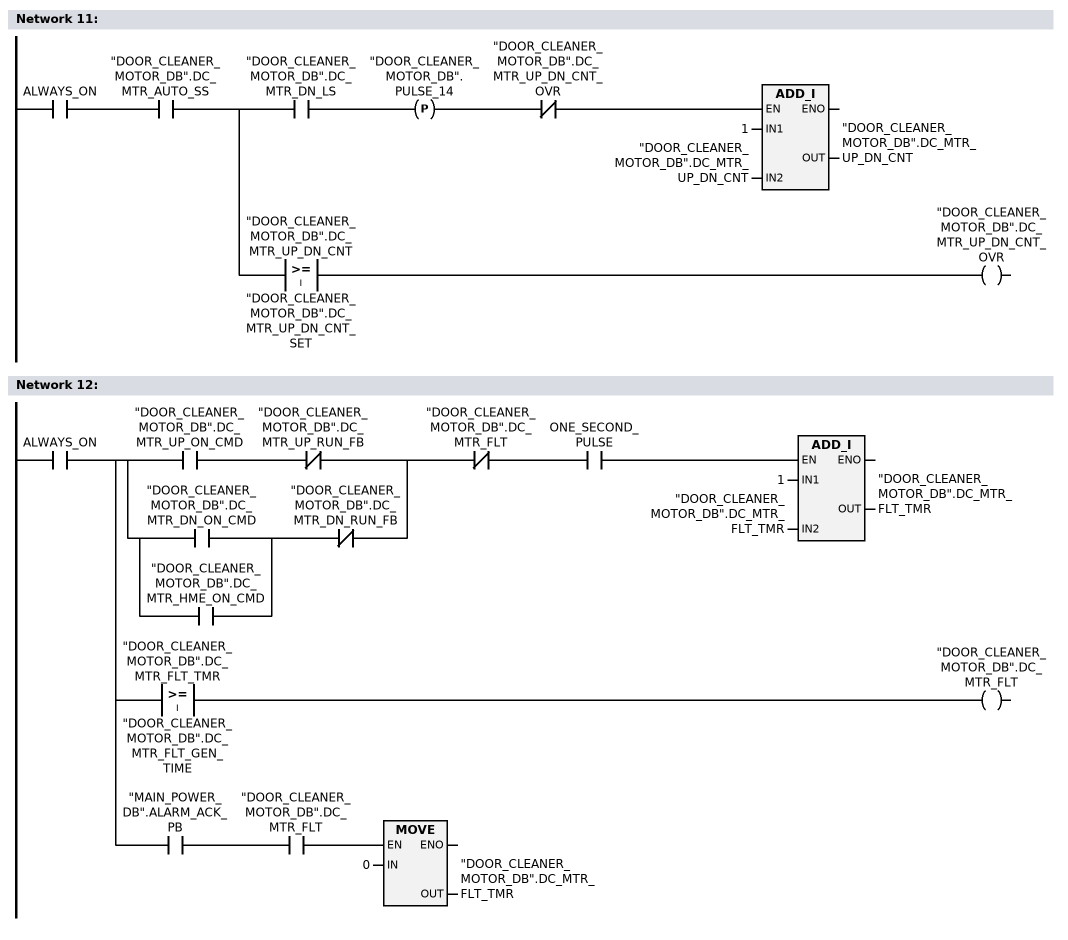
NETWORK
TITLE =
      A     "ALWAYS_ON";
      A     "DOOR_CLEANER_MOTOR_DB".DC_MTR_AUTO_SS;
      =     L 0.0;
      A     L 0.0;
      A     "DOOR_CLEANER_MOTOR_DB".DC_MTR_DN_LS;
      FP    "DOOR_CLEANER_MOTOR_DB".PULSE_14;
      AN    "DOOR_CLEANER_MOTOR_DB".DC_MTR_UP_DN_CNT_OVR;
      JNB   M005;
      L     1;
      L     "DOOR_CLEANER_MOTOR_DB".DC_MTR_UP_DN_CNT;
      +I;
      T     "DOOR_CLEANER_MOTOR_DB".DC_MTR_UP_DN_CNT;
M005: NOP   0;
      A     L 0.0;
      A(;
      L     "DOOR_CLEANER_MOTOR_DB".DC_MTR_UP_DN_CNT;
      L     "DOOR_CLEANER_MOTOR_DB".DC_MTR_UP_DN_CNT_SET;
      >=I;
      );
      =     "DOOR_CLEANER_MOTOR_DB".DC_MTR_UP_DN_CNT_OVR;
NETWORK
TITLE =
      A     "ALWAYS_ON";
      =     L 0.0;
      A     L 0.0;
      A(;
      A     "DOOR_CLEANER_MOTOR_DB".DC_MTR_UP_ON_CMD;
      AN    "DOOR_CLEANER_MOTOR_DB".DC_MTR_UP_RUN_FB;
      O;
      A(;
      O     "DOOR_CLEANER_MOTOR_DB".DC_MTR_DN_ON_CMD;
      O     "DOOR_CLEANER_MOTOR_DB".DC_MTR_HME_ON_CMD;
      );
      AN    "DOOR_CLEANER_MOTOR_DB".DC_MTR_DN_RUN_FB;
      );
      AN    "DOOR_CLEANER_MOTOR_DB".DC_MTR_FLT;
      A     "ONE_SECOND_PULSE";
      JNB   M006;
      L     1;
      L     "DOOR_CLEANER_MOTOR_DB".DC_MTR_FLT_TMR;
      +I;
      T     "DOOR_CLEANER_MOTOR_DB".DC_MTR_FLT_TMR;
M006: NOP   0;
      A     L 0.0;
      A(;
      L     "DOOR_CLEANER_MOTOR_DB".DC_MTR_FLT_TMR;
      L     "DOOR_CLEANER_MOTOR_DB".DC_MTR_FLT_GEN_TIME;
      >=I;
      );
      =     "DOOR_CLEANER_MOTOR_DB".DC_MTR_FLT;
      A     L 0.0;
      A     "MAIN_POWER_DB".ALARM_ACK_PB;
      A     "DOOR_CLEANER_MOTOR_DB".DC_MTR_FLT;
      JNB   M007;
      L     0;
      T     "DOOR_CLEANER_MOTOR_DB".DC_MTR_FLT_TMR;
M007: NOP   0;
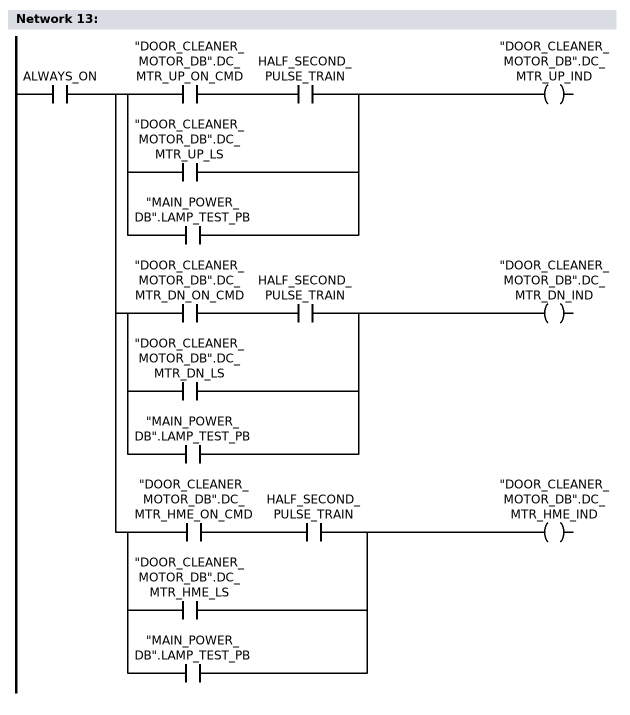
NETWORK
TITLE =
      A     "ALWAYS_ON";
      =     L 0.0;
      A     L 0.0;
      A(;
      A     "DOOR_CLEANER_MOTOR_DB".DC_MTR_UP_ON_CMD;
      A     "HALF_SECOND_PULSE_TRAIN";
      O     "DOOR_CLEANER_MOTOR_DB".DC_MTR_UP_LS;
      O     "MAIN_POWER_DB".LAMP_TEST_PB;
      );
      =     "DOOR_CLEANER_MOTOR_DB".DC_MTR_UP_IND;
      A     L 0.0;
      A(;
      A     "DOOR_CLEANER_MOTOR_DB".DC_MTR_DN_ON_CMD;
      A     "HALF_SECOND_PULSE_TRAIN";
      O     "DOOR_CLEANER_MOTOR_DB".DC_MTR_DN_LS;
      O     "MAIN_POWER_DB".LAMP_TEST_PB;
      );
      =     "DOOR_CLEANER_MOTOR_DB".DC_MTR_DN_IND;
      A     L 0.0;
      A(;
      A     "DOOR_CLEANER_MOTOR_DB".DC_MTR_HME_ON_CMD;
      A     "HALF_SECOND_PULSE_TRAIN";
      O     "DOOR_CLEANER_MOTOR_DB".DC_MTR_HME_LS;
      O     "MAIN_POWER_DB".LAMP_TEST_PB;
      );
      =     "DOOR_CLEANER_MOTOR_DB".DC_MTR_HME_IND;
